	IF T_Data_ProcessImageLoadData.T_GeometryPara.arStartDiameter[6] <> T_Data_ProcessImageData.T_GeometryPara.arStartDiameter[6] THEN xProcessValueModified:=TRUE; RETURN; END_IF
	IF T_Data_ProcessImageLoadData.T_GeometryPara.arEndDiameter[6] <> T_Data_ProcessImageData.T_GeometryPara.arEndDiameter[6] THEN xProcessValueModified:=TRUE; RETURN; END_IF
	IF T_Data_ProcessImageLoadData.T_GeometryPara.arSectionLength[6] <> T_Data_ProcessImageData.T_GeometryPara.arSectionLength[6] THEN xProcessValueModified:=TRUE; RETURN; END_IF
	IF T_Data_ProcessImageLoadData.T_GeometryPara.arSectionPitch[6] <> T_Data_ProcessImageData.T_GeometryPara.arSectionPitch[6] THEN xProcessValueModified:=TRUE; RETURN; END_IF
	IF T_Data_ProcessImageLoadData.T_GeometryPara.axActiveSection[6] <> T_Data_ProcessImageData.T_GeometryPara.axActiveSection[6] THEN xProcessValueModified:=TRUE; RETURN; END_IF
(*09.12.2022: SOA *)
	IF T_Data_ProcessImageLoadData.T_PrismPara.rPrismaDistanceD1 <> T_Data_ProcessImageData.T_PrismPara.rPrismaDistanceD1 THEN xProcessValueModified:=TRUE; RETURN; END_IF
	IF T_Data_ProcessImageLoadData.T_PrismPara.rPrismaDistanceD2 <> T_Data_ProcessImageData.T_PrismPara.rPrismaDistanceD2 THEN xProcessValueModified:=TRUE; RETURN; END_IF
	IF T_Data_ProcessImageLoadData.T_PrismPara.rPrismaAngleA <> T_Data_ProcessImageData.T_PrismPara.rPrismaAngleA THEN xProcessValueModified:=TRUE; RETURN; END_IF
	IF T_Data_ProcessImageLoadData.T_PrismPara.bStateInputPrisma <> T_Data_ProcessImageData.T_PrismPara.bStateInputPrisma THEN xProcessValueModified:=TRUE; RETURN; END_IF
	IF T_Data_ProcessImageLoadData.T_PrismPara.rToolDiameterMin <> T_Data_ProcessImageData.T_PrismPara.rToolDiameterMin THEN xProcessValueModified:=TRUE; RETURN; END_IF
	IF T_Data_ProcessImageLoadData.T_PrismPara.rToolDiameterMax <> T_Data_ProcessImageData.T_PrismPara.rToolDiameterMax THEN xProcessValueModified:=TRUE; RETURN; END_IF
	IF T_Data_ProcessImageLoadData.T_PrismPara.rPrismaFactor <> T_Data_ProcessImageData.T_PrismPara.rPrismaFactor THEN xProcessValueModified:=TRUE; RETURN; END_IF

	IF T_Data_ProcessImageLoadData.T_ProcessPara.rOffsetBeforeToolDiaGrindFeedProcess <> T_Data_ProcessImageData.T_ProcessPara.rOffsetBeforeToolDiaGrindFeedProcess THEN xProcessValueModified:=TRUE; RETURN; END_IF
	IF T_Data_ProcessImageLoadData.T_ProcessPara.rSecurityPosGrindFeedProcess <> T_Data_ProcessImageData.T_ProcessPara.rSecurityPosGrindFeedProcess THEN xProcessValueModified:=TRUE; RETURN; END_IF
	IF T_Data_ProcessImageLoadData.T_ProcessPara.rSpeedBackwardGrindFeed <> T_Data_ProcessImageData.T_ProcessPara.rSpeedBackwardGrindFeed THEN xProcessValueModified:=TRUE; RETURN; END_IF
	IF T_Data_ProcessImageLoadData.T_ProcessPara.rSpeedForwardFastGrindFeed <> T_Data_ProcessImageData.T_ProcessPara.rSpeedForwardFastGrindFeed THEN xProcessValueModified:=TRUE; RETURN; END_IF
	IF T_Data_ProcessImageLoadData.T_ProcessPara.rSpeedForwardSlowGrindFeed <> T_Data_ProcessImageData.T_ProcessPara.rSpeedForwardSlowGrindFeed THEN xProcessValueModified:=TRUE; RETURN; END_IF
	IF xMicroRodActive THEN
		IF T_Data_ProcessImageLoadData.T_ProcessPara.rSpeedStartPosToolFeedProcess <> T_Data_ProcessImageData.T_ProcessPara.rSpeedStartPosToolFeedProcess THEN xProcessValueModified:=TRUE; RETURN; END_IF
		IF T_Data_ProcessImageLoadData.T_ProcessPara.rStartPosToolFeedAuto <> T_Data_ProcessImageData.T_ProcessPara.rStartPosToolFeedAuto THEN xProcessValueModified:=TRUE; RETURN; END_IF
	END_IF;
	IF T_Data_ProcessImageLoadData.T_ProcessPara.rToolDiameterProcess <> T_Data_ProcessImageData.T_ProcessPara.rToolDiameterProcess THEN xProcessValueModified:=TRUE; RETURN; END_IF
	IF T_Data_ProcessImageLoadData.T_ProcessPara.rToolTensionProcess <> T_Data_ProcessImageData.T_ProcessPara.rToolTensionProcess THEN xProcessValueModified:=TRUE; RETURN; END_IF

	IF T_Data_ProcessImageLoadData.T_AutoGeometryPara.iCycleGeometry <> T_Data_ProcessImageData.T_AutoGeometryPara.iCycleGeometry THEN xProcessValueModified:=TRUE; RETURN; END_IF
	IF xMicroRodActive THEN
		IF T_Data_ProcessImageLoadData.T_AutoGeometryPara.rPlungeCycleGrindFeedGeometry <> T_Data_ProcessImageData.T_AutoGeometryPara.rPlungeCycleGrindFeedGeometry THEN xProcessValueModified:=TRUE; RETURN; END_IF
	END_IF;
	IF T_Data_ProcessImageLoadData.T_AutoGeometryPara.rDisplaceLengthToolFeedGeometry <> T_Data_ProcessImageData.T_AutoGeometryPara.rDisplaceLengthToolFeedGeometry THEN xProcessValueModified:=TRUE; RETURN; END_IF
	IF T_Data_ProcessImageLoadData.T_AutoGeometryPara.rDisplaceSpeedGrindFeedGeometry <> T_Data_ProcessImageData.T_AutoGeometryPara.rDisplaceSpeedGrindFeedGeometry THEN xProcessValueModified:=TRUE; RETURN; END_IF
	IF T_Data_ProcessImageLoadData.T_AutoGeometryPara.rPlungeLengthToolFeedGeometry <> T_Data_ProcessImageData.T_AutoGeometryPara.rPlungeLengthToolFeedGeometry THEN xProcessValueModified:=TRUE; RETURN; END_IF
	IF T_Data_ProcessImageLoadData.T_AutoGeometryPara.rPlungeSpeedGrindFeedGeometry <> T_Data_ProcessImageData.T_AutoGeometryPara.rPlungeSpeedGrindFeedGeometry THEN xProcessValueModified:=TRUE; RETURN; END_IF
	IF T_Data_ProcessImageLoadData.T_AutoGeometryPara.rSpeedToolRotationGeometry <> T_Data_ProcessImageData.T_AutoGeometryPara.rSpeedToolRotationGeometry THEN xProcessValueModified:=TRUE; RETURN; END_IF
	IF T_Data_ProcessImageLoadData.T_AutoGeometryPara.xDisplaceActivationGeometry <> T_Data_ProcessImageData.T_AutoGeometryPara.xDisplaceActivationGeometry THEN xProcessValueModified:=TRUE; RETURN; END_IF
	IF T_Data_ProcessImageLoadData.T_AutoGeometryPara.xPlungeActivationGeometry <> T_Data_ProcessImageData.T_AutoGeometryPara.xPlungeActivationGeometry THEN xProcessValueModified:=TRUE; RETURN; END_IF

	IF T_Data_ProcessImageLoadData.T_AutoGroovePara.rDisplaceLengthToolFeedGroove <> T_Data_ProcessImageData.T_AutoGroovePara.rDisplaceLengthToolFeedGroove THEN xProcessValueModified:=TRUE; RETURN; END_IF
	IF T_Data_ProcessImageLoadData.T_AutoGroovePara.rDisplaceSpeedGrindFeedGroove <> T_Data_ProcessImageData.T_AutoGroovePara.rDisplaceSpeedGrindFeedGroove THEN xProcessValueModified:=TRUE; RETURN; END_IF
	IF T_Data_ProcessImageLoadData.T_AutoGroovePara.rPitchGroove <> T_Data_ProcessImageData.T_AutoGroovePara.rPitchGroove THEN xProcessValueModified:=TRUE; RETURN; END_IF
	IF T_Data_ProcessImageLoadData.T_AutoGroovePara.rPlungeLengthToolFeedGroove <> T_Data_ProcessImageData.T_AutoGroovePara.rPlungeLengthToolFeedGroove THEN xProcessValueModified:=TRUE; RETURN; END_IF
	IF T_Data_ProcessImageLoadData.T_AutoGroovePara.rPlungeSpeedGrindFeedGroove <> T_Data_ProcessImageData.T_AutoGroovePara.rPlungeSpeedGrindFeedGroove THEN xProcessValueModified:=TRUE; RETURN; END_IF
	IF T_Data_ProcessImageLoadData.T_AutoGroovePara.rSpeedToolRotationGroove <> T_Data_ProcessImageData.T_AutoGroovePara.rSpeedToolRotationGroove THEN xProcessValueModified:=TRUE; RETURN; END_IF
	IF T_Data_ProcessImageLoadData.T_AutoGroovePara.xDisplaceActivationGroove <> T_Data_ProcessImageData.T_AutoGroovePara.xDisplaceActivationGroove THEN xProcessValueModified:=TRUE; RETURN; END_IF
	IF T_Data_ProcessImageLoadData.T_AutoGroovePara.xPlungeActivationGroove <> T_Data_ProcessImageData.T_AutoGroovePara.xPlungeActivationGroove THEN xProcessValueModified:=TRUE; RETURN; END_IF
	IF T_Data_ProcessImageLoadData.T_AutoGroovePara.xBlockGrindFeeder <> T_Data_ProcessImageData.T_AutoGroovePara.xBlockGrindFeeder THEN xProcessValueModified:=TRUE; RETURN; END_IF
	IF T_Data_ProcessImageLoadData.T_AutoGroovePara.iNumberOfGrooves <> T_Data_ProcessImageData.T_AutoGroovePara.iNumberOfGrooves THEN xProcessValueModified:=TRUE; RETURN; END_IF
	IF T_Data_ProcessImageLoadData.T_AutoGroovePara.iSpeedGrindSpindle <> T_Data_ProcessImageData.T_AutoGroovePara.iSpeedGrindSpindle THEN xProcessValueModified:=TRUE; RETURN; END_IF

	IF T_Data_ProcessImageLoadData.T_CalibrationPara.rDisplaceLengthToolFeedCalib <> T_Data_ProcessImageData.T_CalibrationPara.rDisplaceLengthToolFeedCalib THEN xProcessValueModified:=TRUE; RETURN; END_IF
	IF T_Data_ProcessImageLoadData.T_CalibrationPara.rDisplaceSpeedGrindFeedCalib <> T_Data_ProcessImageData.T_CalibrationPara.rDisplaceSpeedGrindFeedCalib THEN xProcessValueModified:=TRUE; RETURN; END_IF
	IF NOT(xMicroRodActive) THEN
		IF T_Data_ProcessImageLoadData.T_CalibrationPara.rMeasureOffsetToolFeedCalib <> T_Data_ProcessImageData.T_CalibrationPara.rMeasureOffsetToolFeedCalib THEN xProcessValueModified:=TRUE; RETURN; END_IF
	END_IF;
	IF xMicroRodActive THEN
		IF T_Data_ProcessImageLoadData.T_CalibrationPara.rMeasurePosToolFeedCalib <> T_Data_ProcessImageData.T_CalibrationPara.rMeasurePosToolFeedCalib THEN xProcessValueModified:=TRUE; RETURN; END_IF
		IF T_Data_ProcessImageLoadData.T_CalibrationPara.rStartPosToolFeedCalib <> T_Data_ProcessImageData.T_CalibrationPara.rStartPosToolFeedCalib THEN xProcessValueModified:=TRUE; RETURN; END_IF
	END_IF;
	IF T_Data_ProcessImageLoadData.T_CalibrationPara.rPitchCalib <> T_Data_ProcessImageData.T_CalibrationPara.rPitchCalib THEN xProcessValueModified:=TRUE; RETURN; END_IF
	IF T_Data_ProcessImageLoadData.T_CalibrationPara.rPlungeLengthGrindFeedCalib <> T_Data_ProcessImageData.T_CalibrationPara.rPlungeLengthGrindFeedCalib THEN xProcessValueModified:=TRUE; RETURN; END_IF
	IF T_Data_ProcessImageLoadData.T_CalibrationPara.rPlungeLengthToolFeedCalib <> T_Data_ProcessImageData.T_CalibrationPara.rPlungeLengthToolFeedCalib THEN xProcessValueModified:=TRUE; RETURN; END_IF
	IF T_Data_ProcessImageLoadData.T_CalibrationPara.rPlungeSpeedGrindFeedCalib <> T_Data_ProcessImageData.T_CalibrationPara.rPlungeSpeedGrindFeedCalib THEN xProcessValueModified:=TRUE; RETURN; END_IF
	IF T_Data_ProcessImageLoadData.T_CalibrationPara.rSpeedToolRotationCalib <> T_Data_ProcessImageData.T_CalibrationPara.rSpeedToolRotationCalib THEN xProcessValueModified:=TRUE; RETURN; END_IF
	IF T_Data_ProcessImageLoadData.T_CalibrationPara.rToolLengthCylinderPartCalib <> T_Data_ProcessImageData.T_CalibrationPara.rToolLengthCylinderPartCalib THEN xProcessValueModified:=TRUE; RETURN; END_IF
	IF T_Data_ProcessImageLoadData.T_CalibrationPara.xDisplaceActivationCalib <> T_Data_ProcessImageData.T_CalibrationPara.xDisplaceActivationCalib THEN xProcessValueModified:=TRUE; RETURN; END_IF
	IF T_Data_ProcessImageLoadData.T_CalibrationPara.xPlungeActivationCalib <> T_Data_ProcessImageData.T_CalibrationPara.xPlungeActivationCalib THEN xProcessValueModified:=TRUE; RETURN; END_IF
END_FUNCTION_BLOCK

(* POU PRG_VISU_LAYER5/FB_VISU/FB_CALC_TORQUE, ST *)
FUNCTION_BLOCK FB_CALC_TORQUE
VAR_INPUT
	xStart:BOOL;				(* start the calculation of the mean value of the torque *)
	uiActualTorque:UINT;		(* actual current value *)
	uiZeroTorque:UINT;		(* set value of the current value for scale the range *)
	iStepCalc:INT;			(* number of mean value *)
END_VAR
VAR_OUTPUT
	uiCalcTorque:UINT;		(* calculated torque value in % of the maximal torque of the motor *)
END_VAR
VAR
	auiSaveTorque: ARRAY [1..200] OF UINT;
	auiTmpSaveTorque: ARRAY [1..200] OF UINT;
	auiDeleteTorque: ARRAY [1..200] OF UINT;
	uiSumTorque: UINT;
	ii: INT;
	xInit: BOOL;
	uiTmpZeroTorque:UINT;
	rMaxMotorCurrent: REAL;
	rMaxMotorTorque: REAL;
END_VAR
(****************************************************************************************************************************************************)
(***********             This Functionblock calc the torque of the ToolRotation with set and reset torque function                         ************)
(****************************************************************************************************************************************************)
uiCalcTorque:=0;
IF NOT(xStart) AND xInit THEN
	xInit:=FALSE;
	auiSaveTorque:=auiDeleteTorque;
	auiTmpSaveTorque:=auiDeleteTorque;
	uiTmpZeroTorque:=uiZeroTorque;
END_IF;
IF xStart THEN
	xInit:=TRUE;
	uiSumTorque:=0;
	IF (uiZeroTorque <> uiTmpZeroTorque) THEN
		auiSaveTorque:=auiDeleteTorque;
		auiTmpSaveTorque:=auiDeleteTorque;
		uiTmpZeroTorque:=uiZeroTorque;
	END_IF;
	IF (iStepCalc > 0) AND (iStepCalc <= 200) THEN
		FOR ii:=1 TO (iStepCalc - 1)  DO
			auiTmpSaveTorque[ii+1]:=auiSaveTorque[ii];
			uiSumTorque:=uiSumTorque + auiSaveTorque[ii];
		END_FOR;
		auiSaveTorque:=auiTmpSaveTorque;
		IF (uiTmpZeroTorque <= uiActualTorque) THEN
			auiSaveTorque[1]:=uiActualTorque - uiTmpZeroTorque;
		ELSE
			auiSaveTorque[1]:=0;
		END_IF;
		uiSumTorque:=uiSumTorque + auiSaveTorque[1];
		uiSumTorque:=uiSumTorque/iStepCalc;
		rMaxMotorCurrent:=6.0;	(* EcoStep Motor 23S21  *)
		rMaxMotorTorque:=(rMaxMotorCurrent * 0.16) * 1000.0;	(* 0.16 = 0.16Nm/A -->1000.0= Umwandlung in mNm *)
		uiCalcTorque:=REAL_TO_UINT((UINT_TO_REAL(uiSumTorque) / (REAL_TO_UINT(rMaxMotorTorque) - uiTmpZeroTorque)) * 100.0);	(* Ausgabe in % des Max Stromes *)
		IF (uiCalcTorque >= 100) THEN
			uiCalcTorque:=100;
		END_IF;
	END_IF;
END_IF;
END_FUNCTION_BLOCK

(* POU PRG_VISU_LAYER5/FB_VISU/FBQVIS_ERROR_LIST, ST *)
FUNCTION_BLOCK FBQVIS_ERROR_LIST
VAR_INPUT
	T_ErrorList:ST_ERROR_LIST;					(* Static define Error List *)
	T_ErrorNrList:ST_RETAIN_ERROR_DATA;		(* Daten welche im NOVram abgelegt sind *)
END_VAR
VAR_IN_OUT
	T_MsgErrorEnglish:ST_EXCHG_MESSAGE_ERROR;	(* Daten die auf der Visu in der Errorliste visualisiert werden *)
	T_MsgErrorDeutsch:ST_EXCHG_MESSAGE_ERROR;	(* Daten die auf der Visu in der Errorliste visualisiert werden *)
	T_MsgErrorFrancais:ST_EXCHG_MESSAGE_ERROR;	(* Daten die auf der Visu in der Errorliste visualisiert werden *)
END_VAR
VAR_OUTPUT
END_VAR
VAR
	FBErrorMessage:FB_ErrorMessage;
	ii:INT;
	diErrorNr: DINT;
	sErrorTimeStamp: STRING(12);
END_VAR
(****************************************************************************************************************************************************)
(***********                              This Functionblock fills the errorlist with the errormesse and the timestamp                                  ************)
(****************************************************************************************************************************************************)
	FOR ii:=1 TO 20 DO
		diErrorNr:=T_ErrorNrList.adiErrorListMachine[ii];
		sErrorTimeStamp:=T_ErrorNrList.asErrorTimeStampMachine[ii];
		sErrorTimeStamp:=CONCAT(sErrorTimeStamp,'--');
		IF (diErrorNr <> 0) THEN
			FBErrorMessage(	diErrorNr:=diErrorNr ,
							T_ErrorList:=T_ErrorList);
			T_MsgErrorEnglish.asMsgErrorList[ii]:=CONCAT(sErrorTimeStamp,FBErrorMessage.sErrorTextEnglish);
			T_MsgErrorDeutsch.asMsgErrorList[ii]:=CONCAT(sErrorTimeStamp,FBErrorMessage.sErrorTextDeutsch);
			T_MsgErrorFrancais.asMsgErrorList[ii]:=CONCAT(sErrorTimeStamp,FBErrorMessage.sErrorTextFrancais);
		ELSE
			T_MsgErrorEnglish.asMsgErrorList[ii]:='                                                                    ';
			T_MsgErrorDeutsch.asMsgErrorList[ii]:='                                                                    ';
			T_MsgErrorFrancais.asMsgErrorList[ii]:='                                                                    ';
		END_IF;
	END_FOR;
END_FUNCTION_BLOCK

(* POU PRG_VISU_LAYER5/FB_VISU/FB_SETERRORLIST, ST *)
FUNCTION_BLOCK FB_SETERRORLIST
VAR_INPUT
	TControlStation : ST_CONTROL;					(* Control structur of the data station structure *)
	TProcess : ST_PROCESS;						(* data structure of the processlevel *)
END_VAR
VAR_IN_OUT
	xParameterSaved:BOOL;						(* state, if the changed errorlist was saved *)
	T_ErrorNrList:ST_RETAIN_ERROR_DATA;		(* Daten welche im NOVram abgelegt sind *)
	xSetForceError:BOOL;							(* manual input of an error into the error list *)
	diSetForceErrorNr:DINT;						(* manual input of an error number into the error list *)
END_VAR
VAR_OUTPUT
	xSaveParameter:BOOL;						(* save the maked or updated error list into the Novram *)
END_VAR
VAR
	xTmpStation: BOOL;
	xTmpProcess: BOOL;
	iTmpStationNr:INT;
	xBlockProcessProc: BOOL;
	xBlockStationProc: BOOL;
	adiTmpErrorList: ARRAY [1..20] OF DINT;
	asTmpErrorList: ARRAY [1..20] OF STRING(12);
	ii:INT;
	xDataChanged: BOOL;
	xQuitError: BOOL;
	TimerCheckQuitError:TON;
	FBNT_GetTime:NT_GetTime;
	xUpdateProcTimeStamp:BOOL;
	xInitGetTime: BOOL;
END_VAR
(****************************************************************************************************************************************************)
(***********                       This Functionblock manage the machine error, for make and update the errorlist                             ************)
(****************************************************************************************************************************************************)
xTmpStation:=TControlStation.xError AND TControlStation.xActiveStation;
xTmpProcess:=TProcess.xError AND TProcess.xRdy;

IF NOT(xDataChanged) THEN
	IF NOT(TProcess.xEnd) AND TProcess.xError AND NOT(xBlockProcessProc) AND NOT(xBlockStationProc) AND NOT(xSetForceError) THEN
		xBlockProcessProc:=TRUE;
		iTmpStationNr:=0;
	END_IF;
	IF TProcess.xEnd AND xTmpStation AND NOT(xBlockStationProc) AND NOT(xBlockProcessProc) AND NOT(xSetForceError) THEN
		xBlockStationProc:=TRUE;
		iTmpStationNr:=1;
	END_IF;
	IF xBlockProcessProc AND NOT(xQuitError) THEN
		adiTmpErrorList:=T_ErrorNrList.adiErrorListMachine;
		T_ErrorNrList.adiErrorListMachine[1]:=TProcess.diErrorNr;
		FOR ii:=2 TO 20 DO
			T_ErrorNrList.adiErrorListMachine[ii]:=adiTmpErrorList[ii-1];
		END_FOR;
		xUpdateProcTimeStamp:=TRUE;
	END_IF;
	
	IF xBlockStationProc AND NOT(xQuitError) THEN
		adiTmpErrorList:=T_ErrorNrList.adiErrorListMachine;
		T_ErrorNrList.adiErrorListMachine[1]:=TControlStation.diErrorNr;
		FOR ii:=2 TO 20 DO
			T_ErrorNrList.adiErrorListMachine[ii]:=adiTmpErrorList[ii-1];
		END_FOR;
		xUpdateProcTimeStamp:=TRUE;
	END_IF;
	
	IF xSetForceError AND NOT(xQuitError) AND NOT(xBlockStationProc) AND NOT(xBlockProcessProc) THEN
		adiTmpErrorList:=T_ErrorNrList.adiErrorListMachine;
		T_ErrorNrList.adiErrorListMachine[1]:=diSetForceErrorNr;
		FOR ii:=2 TO 20 DO
			T_ErrorNrList.adiErrorListMachine[ii]:=adiTmpErrorList[ii-1];
		END_FOR;
		xUpdateProcTimeStamp:=TRUE;
		xSetForceError:=FALSE;
	ELSE
		xSetForceError:=FALSE;
	END_IF;

	IF xUpdateProcTimeStamp THEN
		IF NOT(xInitGetTime) THEN
			xInitGetTime:=TRUE;
			FBNT_GetTime(	NETID:= '',
							START:=FALSE );
		END_IF;
		FBNT_GetTime(	NETID:= '',
						START:= TRUE,
						TMOUT:= T#2s);
		IF NOT(FBNT_GetTime.BUSY) OR FBNT_GetTime.ERR THEN
			IF xUpdateProcTimeStamp THEN
				asTmpErrorList:=T_ErrorNrList.asErrorTimeStampMachine;
				IF NOT(FBNT_GetTime.ERR) THEN
					T_ErrorNrList.asErrorTimeStampMachine[1]:=Fct_ConvertDateToString(2,FBNT_GetTime.TIMESTR);
				ELSE
					T_ErrorNrList.asErrorTimeStampMachine[1]:='00.00 00:00';	(* Fehler beim lesen der Systemzeit, daher wird ein default-Wert gesetzt *)
				END_IF;
				FOR ii:=2 TO 20 DO
					T_ErrorNrList.asErrorTimeStampMachine[ii]:=asTmpErrorList[ii-1];
				END_FOR;
			END_IF;
			xInitGetTime:=FALSE;
			xUpdateProcTimeStamp:=FALSE;
			xDataChanged:=TRUE;
		END_IF;
	END_IF;
END_IF;

IF xBlockProcessProc OR xBlockStationProc THEN
	xQuitError:=TRUE;
	IF TControlStation.xQuitError OR TProcess.xQuitError THEN
		xBlockProcessProc:=xBlockStationProc:=xSetForceError:=xQuitError:=FALSE;
	END_IF;
	IF NOT(xTmpStation) AND NOT(xTmpProcess) THEN
		TimerCheckQuitError(IN:=TRUE,PT:=T#1s);
		IF TimerCheckQuitError.Q THEN
			TimerCheckQuitError(IN:=FALSE);
			xBlockProcessProc:=xBlockStationProc:=xSetForceError:=xQuitError:=FALSE;
		END_IF;
	ELSE
		TimerCheckQuitError(IN:=FALSE);
	END_IF;
ELSE
	xQuitError:=FALSE;
END_IF;

IF xDataChanged THEN
	xSaveParameter:=TRUE;
	IF xParameterSaved THEN
		xParameterSaved:=xDataChanged:=xSaveParameter:=FALSE;
	END_IF;
END_IF;
END_FUNCTION_BLOCK

(* POU PRG_PROCESS_LAYER4/FB_PROCESS/Fct_ConvertDateToString, ST *)
FUNCTION Fct_ConvertDateToString : STRING
VAR_INPUT
		iFormat:INT;	(* 0=Langes Date-Time Format; 1=Kurzes Date-Time Format; 2=Sehr Kurzes Date-Time Format *)
					(* 0='28.March 2007  08:47:01' *)
					(* 1='28.03.07 08:47' *)
					(* 2='28.03 08:47' *)
		TProcTimeStart:TIMESTRUCT;
END_VAR
VAR
	sTmpData:STRING(255);
	sTmpData1:STRING(255);
	wYear: WORD;
END_VAR
(****************************************************************************************************************************************************)
(***********                                This Functionblock formate a Date and Time String DD:MM HH:MM:SS                                     ************)
(****************************************************************************************************************************************************)
sTmpData:=sTmpData1:='';
IF (iFormat < 0) OR (iFormat > 2) THEN
	sTmpData1:='Wrong Date';
	Fct_ConvertDateToString:=sTmpData1;
	RETURN;
END_IF;
IF (TProcTimeStart.wDay <> 0) THEN
	IF (TProcTimeStart.wDay >= 0) AND (TProcTimeStart.wDay <= 9) THEN
		sTmpData1:=MUX(TProcTimeStart.wDay,'00','01','02','03','04','05','06','07','08','09');
		sTmpData:=CONCAT(sTmpData,sTmpData1);
	ELSE
		sTmpData:=CONCAT(sTmpData,WORD_TO_STRING(TProcTimeStart.wDay));
	END_IF;
	sTmpData:=CONCAT(sTmpData,'.');
ELSE
	sTmpData1:='Wrong Date';
	Fct_ConvertDateToString:=sTmpData1;
	RETURN;
END_IF;
IF (TProcTimeStart.wMonth <> 0) THEN
	IF (iFormat = 0) THEN
		sTmpData1:=MUX(TProcTimeStart.wMonth-1,'January','February','March','April','May','June','July','August','September','October','November','December');
	END_IF;
	IF (iFormat = 1) OR (iFormat = 2) THEN
		sTmpData1:=MUX(TProcTimeStart.wMonth-1,'01','02','03','04','05','06','07','08','09','10','11','12');
	END_IF;
ELSE
	sTmpData1:='Wrong Date';
	Fct_ConvertDateToString:=sTmpData1;
	RETURN;
END_IF;
sTmpData:=CONCAT(sTmpData,sTmpData1);
IF (iFormat = 0) THEN
	sTmpData:=CONCAT(sTmpData,' ');
END_IF;
IF (iFormat = 1) THEN
	sTmpData:=CONCAT(sTmpData,'.');
END_IF;
IF (iFormat = 2) THEN
	sTmpData:=CONCAT(sTmpData,' ');
END_IF;
IF (iFormat = 0) OR (iFormat = 1) THEN
	IF (TProcTimeStart.wYear <> 0) THEN
		IF (iFormat = 0) THEN
			sTmpData:=CONCAT(sTmpData,WORD_TO_STRING(TProcTimeStart.wYear));
			sTmpData:=CONCAT(sTmpData,'  ');
		END_IF;
		IF (iFormat = 1) THEN
			IF (TProcTimeStart.wYear >= 1000) AND (TProcTimeStart.wYear < 2000) THEN
				wYear:=TProcTimeStart.wYear - 1000;
			END_IF;
			IF (TProcTimeStart.wYear >= 2000) AND (TProcTimeStart.wYear < 3000) THEN
				wYear:=TProcTimeStart.wYear - 2000;
			END_IF;
			IF (wYear >= 0) AND (wYear < 10) THEN
				sTmpData1:=MUX(wYear,'00','01','02','03','04','05','06','07','08','09');
				sTmpData:=CONCAT(sTmpData,sTmpData1);
			ELSE
				sTmpData:=CONCAT(sTmpData,WORD_TO_STRING(wYear));
			END_IF;
			sTmpData:=CONCAT(sTmpData,' ');
		END_IF;
	ELSE
		sTmpData1:='Wrong Date';
		Fct_ConvertDateToString:=sTmpData1;
		RETURN;
	END_IF;
END_IF;
IF (TProcTimeStart.wHour >= 0) AND (TProcTimeStart.wHour <= 9) THEN
	sTmpData1:=MUX(TProcTimeStart.wHour,'00','01','02','03','04','05','06','07','08','09');
	sTmpData:=CONCAT(sTmpData,sTmpData1);
ELSE
	sTmpData:=CONCAT(sTmpData,WORD_TO_STRING(TProcTimeStart.wHour));
END_IF;
sTmpData:=CONCAT(sTmpData,':');
IF (TProcTimeStart.wMinute >= 0) AND (TProcTimeStart.wMinute <= 9) THEN
	sTmpData1:=MUX(TProcTimeStart.wMinute,'00','01','02','03','04','05','06','07','08','09');
	sTmpData:=CONCAT(sTmpData,sTmpData1);
ELSE
	sTmpData:=CONCAT(sTmpData,WORD_TO_STRING(TProcTimeStart.wMinute));
END_IF;
IF (iFormat = 0) THEN
	sTmpData:=CONCAT(sTmpData,':');
	IF (TProcTimeStart.wSecond >= 0) AND (TProcTimeStart.wSecond <= 9) THEN
		sTmpData1:=MUX(TProcTimeStart.wSecond,'00','01','02','03','04','05','06','07','08','09');
		sTmpData:=CONCAT(sTmpData,sTmpData1);
	ELSE
		sTmpData:=CONCAT(sTmpData,WORD_TO_STRING(TProcTimeStart.wSecond));
	END_IF;
END_IF;
Fct_ConvertDateToString:=sTmpData;
END_FUNCTION

(* POU PRG_VISU_LAYER5/FB_VISU/FBQVIS_CLEARERROR, ST *)
FUNCTION_BLOCK FBQVIS_CLEARERROR
VAR_INPUT
	xExecute:BOOL;				(* quit the error *)
	iError:INT;					(* occured error number *)
END_VAR
VAR_IN_OUT
	T_Message:ST_EXCHG_MESSAGE;		(* data structure for the message handling *)
	T_Station:ST_STATION;				(* data structure for the stationlevel *)
	T_Process : ST_PROCESS;			(* data structure for the processlevel *)
	T_NovRAM:ST_NOVRAM;				(* data structure for the Novram *)
	T_Profile:ST_PROFILE;				(* data structure for the profile management *)
	T_HDD:ST_HDD;						(* data structure for the file management *)
END_VAR
VAR_OUTPUT
	xDone:BOOL;
	xNotReady:BOOL;
	xErr:BOOL;
	udiErrorID:UDINT;
END_VAR
VAR
(* Trigger *)
	RisingEdgeExecute:R_TRIG;
(* Pointer *)
	ptrActivStation:POINTER TO ST_STATION;
(* Variable *)
	xClearError_Done:BOOL;
	xClearError_Err:BOOL;
	xClearError_NotReady:BOOL;
	xStepClearDone:BOOL;
	udiClearError_ErrorID:UDINT;
	iStepClearErrorStation:INT;
	iStepClearErrorMachine:INT;
	iStepClearStandardError: INT;
	xClearProcess:BOOL;
	xClearStation:BOOL;
	xClearStandardError:BOOL;
	xClearConifgErrStation: BOOL;
	xTmp: BOOL;
	xClearAxis: BOOL;
	iStepClearErrorAxis: INT;
	xTmp1: BOOL;
	xActiveMicroRod: BOOL;
	iTryAgain: INT;
END_VAR
(****************************************************************************************************************************************************)
(***********              This Functionblock manage an occured machine error so that the right component are quittet              ************)
(****************************************************************************************************************************************************)
	IF (T_NovRAM.T_Data.T_Standard.T_MachineConfig.iConfigMachineType = 2) THEN
		xActiveMicroRod:=TRUE;
	ELSE
		xActiveMicroRod:=FALSE;
	END_IF;

	RisingEdgeExecute(CLK:=xExecute);
	IF RisingEdgeExecute.Q THEN
	(* Init. variable by start clear error *)
		(* ...output *)
		xDone:=FALSE;
		xNotReady:=FALSE;
		xErr:=FALSE;
		udiErrorID:=16#0;
		(* ...variable *)
		xClearError_Done:=FALSE;
		xClearError_Err:=FALSE;
		xClearError_NotReady:=FALSE;
		xStepClearDone:=FALSE;
		iStepClearErrorStation:=1;
		iStepClearErrorMachine:=1;
		iStepClearStandardError:=1;
		iStepClearErrorAxis:=1;
		(* determin clear action *)
		xClearProcess:=xClearStation:=xClearAxis:=xClearStandardError:=FALSE;
		xClearConifgErrStation:=FALSE;
		IF T_Process.xError THEN
			xClearProcess:=TRUE;
		ELSE
			IF T_Station.TControl.xError AND NOT(T_Station.TControl.xEnd) THEN ptrActivStation:=ADR(T_Station); xClearStation:=TRUE; END_IF
			xTmp:=	(T_Station.THardware.TAxisToolLeft.T_CtrleSingle.xErr OR
					(T_Station.THardware.TAxisToolCenter.T_CtrleSingle.xErr AND xActiveMicroRod) OR
					T_Station.THardware.TAxisToolRight.T_CtrleSingle.xErr OR
					T_Station.THardware.TAxisToolFeeder.T_CtrleSingle.xErr OR
					T_Station.THardware.TAxisGrindFeeder.T_CtrleSingle.xErr) AND
					NOT(xClearStation);
			IF xTmp THEN
				xClearAxis:=TRUE;
			END_IF;
			IF T_Station.TControl.xError AND T_Station.TControl.xEnd AND NOT(xClearAxis) THEN
				xClearConifgErrStation:=TRUE;
			END_IF
		END_IF
		IF NOT xClearProcess AND NOT xClearStation AND NOT xClearConifgErrStation AND NOT xClearAxis THEN xClearStandardError:=TRUE; END_IF
		(* Exit FB *)
		RETURN;
	END_IF

	IF xClearProcess THEN
	(* Reset Error machine *)
		CASE iStepClearErrorMachine OF
		(* check station *)
		1:	IF T_Process.xError THEN iStepClearErrorMachine:=10; ELSE iStepClearErrorMachine:=90; END_IF
		(* activ clear error *)
		10:	T_Process.xQuitError:=TRUE;
			(* next step *)
			iStepClearErrorMachine:=20;
			xStepClearDone:=FALSE;
		(* waiting end clearing error *)
		20:	IF NOT T_Process.xQuitError THEN
				iStepClearErrorMachine:=90;
				xStepClearDone:=FALSE;
			END_IF
			IF T_Process.xError THEN iStepClearErrorMachine:=90; END_IF
		(* Clear error station done *)
		90:	xClearError_Done:=TRUE;
		(* Error *)
		99:	xClearError_Err:=TRUE;
		END_CASE
	END_IF

	IF xClearStation THEN
	(* Reset Error station *)
		CASE iStepClearErrorStation OF
		(* check station *)
		1:	IF ptrActivStation^.TControl.xError THEN iStepClearErrorStation:=10;
			ELSE IStepClearErrorStation:=90; END_IF
		(* activ clear error *)
		10:	ptrActivStation^.TControl.xQuitError:=TRUE;
			(* next step *)
			iStepClearErrorStation:=20;
			xStepClearDone:=FALSE;
		(* waiting end clearing error *)
		20:	IF NOT(xStepClearDone) THEN
			(* release action *)
				ptrActivStation^.TControl.xQuitError:=FALSE;
				xStepClearDone:=TRUE;
			ELSE
				IF ptrActivStation^.TControl.xEnd THEN
				(* confirm clear error, next step *)
					iStepClearErrorStation:=90;
					xStepClearDone:=FALSE;
				END_IF
				IF ptrActivStation^.TControl.xError THEN iStepClearErrorStation:=99; END_IF
			END_IF
		(* Clear error station done *)
		90:	xClearError_Done:=TRUE;
		(* Error *)
		99:	xClearError_Done:=TRUE;
		END_CASE
	END_IF

	IF xClearConifgErrStation THEN
		T_Station.TControl.xError:=FALSE;
		xClearConifgErrStation:=FALSE;
		(* Clear error station done *)
		xClearError_Done:=TRUE;
	END_IF;

	IF xClearAxis THEN
	(* Reset Error axis *)
		CASE iStepClearErrorAxis OF
		(* check station *)
		1:	xTmp:=	T_Station.THardware.TAxisToolLeft.T_CtrleSingle.xErr OR
					(T_Station.THardware.TAxisToolCenter.T_CtrleSingle.xErr AND xActiveMicroRod) OR
					T_Station.THardware.TAxisToolRight.T_CtrleSingle.xErr OR
					T_Station.THardware.TAxisToolFeeder.T_CtrleSingle.xErr OR
					T_Station.THardware.TAxisGrindFeeder.T_CtrleSingle.xErr;
			IF xTmp THEN iStepClearErrorAxis:=10;
			ELSE iStepClearErrorAxis:=90; END_IF
			iTryAgain:=0;
		(* activ clear error *)
		10:	T_Station.THardware.TAxisToolLeft.T_CtrleSingle.iFunction:=1;
			T_Station.THardware.TAxisToolLeft.T_CtrleSingle.xExecute:=T_Station.THardware.TAxisToolLeft.T_CtrleSingle.xErr;
			IF xActiveMicroRod THEN
				T_Station.THardware.TAxisToolCenter.T_CtrleSingle.iFunction:=1;
				T_Station.THardware.TAxisToolCenter.T_CtrleSingle.xExecute:=T_Station.THardware.TAxisToolCenter.T_CtrleSingle.xErr;
			END_IF;
			T_Station.THardware.TAxisToolRight.T_CtrleSingle.iFunction:=1;
			T_Station.THardware.TAxisToolRight.T_CtrleSingle.xExecute:=T_Station.THardware.TAxisToolRight.T_CtrleSingle.xErr;
			T_Station.THardware.TAxisToolFeeder.T_CtrleSingle.iFunction:=1;
			T_Station.THardware.TAxisToolFeeder.T_CtrleSingle.xExecute:=T_Station.THardware.TAxisToolFeeder.T_CtrleSingle.xErr;
			T_Station.THardware.TAxisGrindFeeder.T_CtrleSingle.iFunction:=1;
			T_Station.THardware.TAxisGrindFeeder.T_CtrleSingle.xExecute:=T_Station.THardware.TAxisGrindFeeder.T_CtrleSingle.xErr;
			(* next step *)
			iStepClearErrorAxis:=20;
			xStepClearDone:=FALSE;
		(* waiting end clearing error *)
		20:	IF NOT(xStepClearDone) THEN
			(* release action *)
				xStepClearDone:=TRUE;
			ELSE
				xTmp:=	T_Station.THardware.TAxisToolLeft.T_CtrleSingle.xDone AND
						((T_Station.THardware.TAxisToolCenter.T_CtrleSingle.xDone AND xActiveMicroRod) OR NOT(xActiveMicroRod)) AND
						T_Station.THardware.TAxisToolRight.T_CtrleSingle.xDone AND
						T_Station.THardware.TAxisToolFeeder.T_CtrleSingle.xDone AND
						T_Station.THardware.TAxisGrindFeeder.T_CtrleSingle.xDone;
				xTmp1:=	T_Station.THardware.TAxisToolLeft.T_CtrleSingle.xErr OR
						(T_Station.THardware.TAxisToolCenter.T_CtrleSingle.xErr AND xActiveMicroRod) OR
						T_Station.THardware.TAxisToolRight.T_CtrleSingle.xErr OR
						T_Station.THardware.TAxisToolFeeder.T_CtrleSingle.xErr OR
						T_Station.THardware.TAxisGrindFeeder.T_CtrleSingle.xErr;
				IF xTmp THEN
				(* confirm clear error, next step *)
					iStepClearErrorAxis:=90;
					xStepClearDone:=FALSE;
				END_IF
				IF xTmp1 THEN
					iTryAgain:=iTryAgain + 1;
					IF (iTryAgain <= 3) THEN
						(* Reset maximal three times *)
						iStepClearErrorAxis:=10;
					ELSE
						iStepClearErrorAxis:=99;
					END_IF;
				END_IF

			END_IF
		(* Clear error station done *)
		90:	xClearError_Done:=TRUE;
		(* Error *)
		99:	xClearError_Done:=TRUE;
		END_CASE;
	END_IF;

	IF xClearStandardError THEN
	(* Reset Error standard *)
		CASE iStepClearStandardError OF
		(* check NovRAM state *)
		1:	iStepClearStandardError:=10;
			IF T_NovRAM.T_Ctrle.xErr THEN T_NovRAM.T_Ctrle.xReset:=TRUE; END_IF
		(* check Profile State *)
		10:	iStepClearStandardError:=20;
			IF T_Profile.T_Ctrle.xErr THEN T_Profile.T_Ctrle.xReset:=TRUE; END_IF
		(* check HDD state *)
		20:	iStepClearStandardError:=90;
			IF T_HDD.T_Ctrle.xErr THEN T_HDD.T_Ctrle.xReset:=TRUE; END_IF
		(* Clear error station done *)
		90:	xClearError_Done:=TRUE;
		END_CASE
	END_IF

(* FB Done/Err/NotReady *)
	IF xClearError_Done OR xClearError_Err OR xClearError_NotReady THEN
	(* copy value *)
		T_Message.iState:=0;
		T_Message.sDynamicTextEnglish:='';
		T_Message.sDynamicTextDeutsch:='';
		T_Message.sDynamicTextFrancais:='';
		xDone:=xClearError_Done;
		xNotReady:=xClearError_NotReady;
		xErr:=FALSE;
		udiErrorID:=udiClearError_ErrorID;
		(* Init. function state *)
		xClearProcess:=FALSE;
		xClearStation:=FALSE;
		xClearAxis:=FALSE;
		xClearStandardError:=FALSE;
		xClearConifgErrStation:=FALSE;
	END_IF
END_FUNCTION_BLOCK

(* POU GENERAL/FB_CALCPROCESSTIME, ST *)
FUNCTION_BLOCK FB_CALCPROCESSTIME
VAR_INPUT
	T_Geometry:ST_GEOMETRY;									(* Structure of the NovRAM parameter *)
	T_AutoGeometryPara:ST_EXCHG_PARAM_AUTOGEOMETRY;		(* Structure of the NovRAM parameter *)
	T_CalibrationPara:ST_EXCHG_PARAM_CALIBRATION;			(* Structure of the NovRAM parameter *)
	T_AutoGroovePara:ST_EXCHG_PARAM_AUTOGROOVE;			(* Structure of the NovRAM parameter *)
	T_ProcessPara:ST_EXCHG_PARAM_PROCESS;					(* Structure of the NovRAM parameter *)
	rToolRotationSpeed:REAL;										(* Speed of the ToolRotation in U/Min *)
	rToolDiameter:REAL;											(* Diameter of the Tool in um *)
	rToolDiameterWithOffset:REAL;			(* diameter of the unworked Tool plus the offset for plunge and displace procedure *)
	iAutoProcess:INT;												(* 0=Calibration, 1=AutoGeometry process, 2=AutoGroove process *)
	xMicroRodActive:BOOL;										(* choice of the machine MicroWire or MicroRod *)
END_VAR
VAR_IN_OUT
	T_WorkTool:ST_WORKTOOL;									(* Tool parameter *)
END_VAR
VAR_OUTPUT
	rProcessTime: REAL;											(* calculated process time *)
END_VAR
VAR
	FBToolCalcul:FB_TOOL_CALCUL;
	ii: INT;
	rTimeLeftWork: REAL;
	iStartSection: INT;
	iEndSection: INT;
	rPlungeGrind: REAL;
	rDisplaceGrind: REAL;
	rGrindFeederPlunge: REAL;
	xResetFB: BOOL;
	xInitFB:BOOL;
(*11.10.2010 KFS {	*)
	FBCalcPlungeGrinding: FB_CALC_PLUNGE_GRINDING;
	FBCalcPlungeGrindingMultiCycle: FB_CALC_PLUNGE_GRINDING_MultiCycle;
(*11.10.2010 KFS }	*)
	rPlungeCycleGrindFeedGeometry: REAL;
	iTmpStartSection: INT;
	xCalculation: BOOL;
	rToolFeedLength: REAL;
	rSpeedToolFeed: REAL;
	rTimeAddLeftWork:REAL;
	rToolLength:REAL;
	rPlungeGrind2: REAL;
	rTimeAddLeftWorkPlungeGrind: REAL;
	rTimeAddLeftWorkPlungeGrind2: REAL;
	rTimeAddLeftWorkToolFeed: REAL;
END_VAR
(****************************************************************************************************************************************************)
(***********        This Functionblock calculates the time,  needed to work a geometry, groove or  calibration      		    ************)
(****************************************************************************************************************************************************)
	rProcessTime:=0.0;
	rTimeLeftWork:=0;
	iStartSection:=0;
	iEndSection:=0;
	xInitFB:=FALSE;
	IF (iAutoProcess = 1) THEN
	(* calculate the time for the process AutoGeometry or AutoGroove *)
		T_WorkTool.iTotalCountDownPlungeCycle:=0;
		(* Check Start and End Section of the ToolGeometry *)
		FOR ii:=1 TO 6 DO
			IF T_Geometry.axActiveSection[ii] THEN
				IF (iStartSection = 0) THEN
					iStartSection:=ii;
				END_IF;
				iEndSection:=ii;
			END_IF;
		END_FOR;
		xResetFB:=TRUE;
		(* reset first the FB for calculate the grinding plunge for each sections *)
		FBCalcPlungeGrindingMultiCycle(	rToolDiameter:= rToolDiameter,
										rToolDiameterWithOffset:=rToolDiameterWithOffset,
										xReset:= xResetFB,
										xInit:=xInitFB);
		xInitFB:=TRUE;
		FBCalcPlungeGrindingMultiCycle(	T_Geometry:= T_Geometry,
										T_AutoGeometryPara:= T_AutoGeometryPara,
										rToolDiameter:= rToolDiameter,
										rToolDiameterWithOffset:=rToolDiameterWithOffset,
										rPlungeCycleGrindFeedGeometry:=rPlungeCycleGrindFeedGeometry,
										iStartSection:= iStartSection,
										iEndSection:= iEndSection,
										xReset:= xResetFB,
										xInit:=xInitFB);

		rPlungeCycleGrindFeedGeometry:=1.0;
		IF (iAutoProcess = 1) AND xMicroRodActive THEN
			rPlungeCycleGrindFeedGeometry:=T_AutoGeometryPara.rPlungeCycleGrindFeedGeometry;
		END_IF;
		T_WorkTool.rToolRotationSpeed:=rToolRotationSpeed;
		xCalculation:=TRUE;
		WHILE(xCalculation) DO
			(* calculate the grinding way of each section *)
			FBCalcPlungeGrindingMultiCycle(	T_Geometry:= T_Geometry,
											T_AutoGeometryPara:= T_AutoGeometryPara,
											rToolDiameter:= rToolDiameter,
											rToolDiameterWithOffset:=rToolDiameterWithOffset,
											rPlungeCycleGrindFeedGeometry:=rPlungeCycleGrindFeedGeometry,
											iStartSection:= iStartSection,
											iEndSection:= iEndSection,
											xReset:= xResetFB,
											xInit:=xInitFB);
			IF FBCalcPlungeGrindingMultiCycle.xEndWorking THEN		(* check if the end of the to work Tool is reached *)
				xCalculation:=FALSE;
				EXIT;
			END_IF;
			IF (FBCalcPlungeGrindingMultiCycle.iStepSectionWork = 7) THEN
				(* Count the Plunge Cycle *)
				T_WorkTool.iTotalCountDownPlungeCycle:=T_WorkTool.iTotalCountDownPlungeCycle + 1;
			END_IF;
			IF (FBCalcPlungeGrindingMultiCycle.iStepSectionWork >= 1) AND (FBCalcPlungeGrindingMultiCycle.iStepSectionWork <= 6) THEN
			(* section 1 - 6 *)
				iTmpStartSection:=iStartSection + (FBCalcPlungeGrindingMultiCycle.iStepSectionWork - 1);
				rGrindFeederPlunge:=FBCalcPlungeGrindingMultiCycle.rGrindingRelativePosition;
				T_WorkTool.rGrindFeederPlunge:=rGrindFeederPlunge;
				T_WorkTool.rPitch:=T_Geometry.arSectionPitch[iTmpStartSection];
				T_WorkTool.rToolLength:=T_Geometry.arSectionLength[iTmpStartSection];
				FBToolCalcul(	xMicroRodActive:=xMicroRodActive,
								xBeckhoffDriveActive:=FALSE,
								T_WorkTool:= T_WorkTool);
				rTimeLeftWork:=rTimeLeftWork + T_WorkTool.rTimeLeftWork;
			END_IF;
			IF (FBCalcPlungeGrindingMultiCycle.iStepSectionWork = 0) THEN
				(* Calc Plunge *)
				IF T_AutoGeometryPara.xPlungeActivationGeometry THEN
					T_WorkTool.rPitch:=T_Geometry.arSectionPitch[iStartSection] * -1.0;
					T_WorkTool.rGrindFeederPlunge:=FBCalcPlungeGrindingMultiCycle.rGrindingRelativePosition;
					rToolFeedLength:=T_AutoGeometryPara.rPlungeLengthToolFeedGeometry;
					T_WorkTool.rToolLength:=rToolFeedLength;
					T_WorkTool.rToolRotationSpeed:=T_AutoGeometryPara.rSpeedToolRotationGeometry;
					FBToolCalcul(	xMicroRodActive:=xMicroRodActive,
									xBeckhoffDriveActive:=FALSE,
									T_WorkTool:= T_WorkTool);
					rSpeedToolFeed:=T_WorkTool.rToolFeederSpeedUnit * -1.0;
					IF (rSpeedToolFeed <> 0) THEN
						rTimeLeftWork:=rTimeLeftWork + T_WorkTool.rToolLength/rSpeedToolFeed;
					END_IF;
				ELSE
					(* No Plunging activation, than also is the GrindFeeder the master *)
					rPlungeGrind:=ABS(FBCalcPlungeGrindingMultiCycle.rGrindingRelativePosition);
					IF (T_AutoGeometryPara.rPlungeSpeedGrindFeedGeometry <> 0) THEN
						rTimeLeftWork:=rTimeLeftWork + (rPlungeGrind / T_AutoGeometryPara.rPlungeSpeedGrindFeedGeometry);
					END_IF;
				END_IF;
			END_IF;
			IF (FBCalcPlungeGrindingMultiCycle.iStepSectionWork = 7) THEN
				(* Calc Displace *)
				IF T_AutoGeometryPara.xDisplaceActivationGeometry THEN
					T_WorkTool.rPitch:=T_Geometry.arSectionPitch[iEndSection] * -1.0;
					T_WorkTool.rGrindFeederPlunge:=FBCalcPlungeGrindingMultiCycle.rGrindingRelativePosition;
					rToolFeedLength:=T_AutoGeometryPara.rDisplaceLengthToolFeedGeometry;
					T_WorkTool.rToolLength:=rToolFeedLength;
					T_WorkTool.rToolRotationSpeed:=T_AutoGeometryPara.rSpeedToolRotationGeometry;
					FBToolCalcul(	xMicroRodActive:=xMicroRodActive,
									xBeckhoffDriveActive:=FALSE,
									T_WorkTool:= T_WorkTool);
					rSpeedToolFeed:=T_WorkTool.rToolFeederSpeedUnit * -1.0;
					IF (rSpeedToolFeed <> 0) THEN
						rTimeLeftWork:=rTimeLeftWork + T_WorkTool.rToolLength/rSpeedToolFeed;
					END_IF;
				ELSE
					(* No Displace activation, than also is the GrindFeeder the master *)
					rDisplaceGrind:=ABS(FBCalcPlungeGrindingMultiCycle.rGrindingRelativePosition);
					IF (T_AutoGeometryPara.rDisplaceSpeedGrindFeedGeometry <> 0) THEN
						rTimeLeftWork:=rTimeLeftWork + (rDisplaceGrind / T_AutoGeometryPara.rDisplaceSpeedGrindFeedGeometry);
					END_IF;
				END_IF;
			END_IF;
		END_WHILE;
		IF (T_AutoGeometryPara.iCycleGeometry > 1) THEN
			rTimeLeftWork:=rTimeLeftWork * INT_TO_REAL(T_AutoGeometryPara.iCycleGeometry);
		END_IF;
	END_IF;
(**************iAutoProcess 2 --> AutoGroove********************************************************************************************************************************************************************************************************)
	IF (iAutoProcess = 2) THEN
	(* calculate the time for the process AutoGeometry or AutoGroove *)
		T_WorkTool.iTotalCountDownPlungeCycle:=0;
		(* Check Start and End Section of the ToolGeometry *)
		FOR ii:=1 TO 6 DO
			IF T_Geometry.axActiveSection[ii] THEN
				IF (iStartSection = 0) THEN
					iStartSection:=ii;
				END_IF;
				iEndSection:=ii;
			END_IF;
		END_FOR;
(*
		xResetFB:=TRUE;
		(* reset first the FB for calculate the grinding plunge for each sections *)
		FBCalcPlungeGrinding(	rToolDiameter:= rToolDiameter,
								rToolDiameterWithOffset:=rToolDiameterWithOffset,
								xReset:= xResetFB);
		rPlungeCycleGrindFeedGeometry:=1.0;
*)
		xResetFB:=TRUE;
		(* reset first the FB for calculate the grinding plunge for each sections *)
		FBCalcPlungeGrindingMultiCycle(	rToolDiameter:= rToolDiameter,
										rToolDiameterWithOffset:=rToolDiameterWithOffset,
										xReset:= xResetFB,
										xInit:=xInitFB);
		xInitFB:=TRUE;
		FBCalcPlungeGrindingMultiCycle(	T_Geometry:= T_Geometry,
										T_AutoGeometryPara:= T_AutoGeometryPara,
										rToolDiameter:= rToolDiameter,
										rToolDiameterWithOffset:=rToolDiameterWithOffset,
										rPlungeCycleGrindFeedGeometry:=rPlungeCycleGrindFeedGeometry,
										iStartSection:= iStartSection,
										iEndSection:= iEndSection,
										xReset:= xResetFB,
										xInit:=xInitFB);
		rPlungeCycleGrindFeedGeometry:=1.0;
		IF (iAutoProcess = 2) OR NOT(xMicroRodActive) THEN
			rPlungeCycleGrindFeedGeometry:=rToolDiameter;		(* for the groove process or for the MicroWire is not possible to work in more cycle, because of that it will set the tooldiamter *)
		END_IF;
		T_WorkTool.rToolRotationSpeed:=rToolRotationSpeed;
		xCalculation:=TRUE;
		WHILE(xCalculation) DO
			(* calculate the grinding way of each section *)
			FBCalcPlungeGrindingMultiCycle(	T_Geometry:= T_Geometry,
											T_AutoGeometryPara:= T_AutoGeometryPara,
											rToolDiameter:= rToolDiameter,
											rToolDiameterWithOffset:=rToolDiameterWithOffset,
											rPlungeCycleGrindFeedGeometry:=rPlungeCycleGrindFeedGeometry,
											iStartSection:= iStartSection,
											iEndSection:= iEndSection,
											xReset:= xResetFB,
											xInit:=xInitFB);
			IF FBCalcPlungeGrindingMultiCycle.xEndWorking THEN		(* check if the end of the to work Tool is reached *)
				xCalculation:=FALSE;
				EXIT;
			END_IF;
			IF (T_WorkTool.iTotalCountDownPlungeCycle >= 20) THEN	(* not possible to work a Tool in more that 20 cycle *)
				xCalculation:=FALSE;
				EXIT;
			END_IF;
			IF (FBCalcPlungeGrindingMultiCycle.iStepSectionWork = 7) THEN
				(* Count the Plunge Cycle *)
				T_WorkTool.iTotalCountDownPlungeCycle:=T_WorkTool.iTotalCountDownPlungeCycle + 1;
			END_IF;
			IF (FBCalcPlungeGrindingMultiCycle.iStepSectionWork >= 1) AND (FBCalcPlungeGrindingMultiCycle.iStepSectionWork <= 6) THEN
			(* section 1 - 6 *)
				iTmpStartSection:=iStartSection + (FBCalcPlungeGrindingMultiCycle.iStepSectionWork - 1);
				rGrindFeederPlunge:=FBCalcPlungeGrindingMultiCycle.rGrindingRelativePosition;
				T_WorkTool.rGrindFeederPlunge:=rGrindFeederPlunge;
				T_WorkTool.rPitch:=T_AutoGroovePara.rPitchGroove;
				T_WorkTool.rToolLength:=T_Geometry.arSectionLength[iTmpStartSection];
				FBToolCalcul(	xMicroRodActive:=xMicroRodActive,
								xBeckhoffDriveActive:=FALSE,
								T_WorkTool:= T_WorkTool);
				rTimeLeftWork:=rTimeLeftWork + T_WorkTool.rTimeLeftWork;
			END_IF;
			IF (FBCalcPlungeGrindingMultiCycle.iStepSectionWork = 0) THEN
				(* Calc Plunge *)
				IF T_AutoGroovePara.xPlungeActivationGroove  THEN
					T_WorkTool.rPitch:=T_AutoGroovePara.rPitchGroove * -1.0;
					T_WorkTool.rGrindFeederPlunge:=FBCalcPlungeGrindingMultiCycle.rGrindingRelativePosition;
					rToolFeedLength:=T_AutoGroovePara.rPlungeLengthToolFeedGroove;
					T_WorkTool.rToolLength:=rToolFeedLength;
					T_WorkTool.rToolRotationSpeed:=T_AutoGroovePara.rSpeedToolRotationGroove;
					FBToolCalcul(	xMicroRodActive:=xMicroRodActive,
									xBeckhoffDriveActive:=FALSE,
									T_WorkTool:= T_WorkTool);
					rSpeedToolFeed:=T_WorkTool.rToolFeederSpeedUnit * -1.0;
					IF (rSpeedToolFeed <> 0) THEN
						rTimeLeftWork:=rTimeLeftWork + T_WorkTool.rToolLength/rSpeedToolFeed;
					END_IF;
				ELSE
					(* No Plunging activation, than also is the GrindFeeder the master *)
					rPlungeGrind:=ABS(FBCalcPlungeGrindingMultiCycle.rGrindingRelativePosition);
					IF (T_AutoGroovePara.rPlungeSpeedGrindFeedGroove <> 0) THEN
						rTimeLeftWork:=rTimeLeftWork + (rPlungeGrind / T_AutoGroovePara.rPlungeSpeedGrindFeedGroove);
					END_IF;
				END_IF;
			END_IF;
			IF (FBCalcPlungeGrindingMultiCycle.iStepSectionWork = 7) THEN
				(* Calc Displace *)
				IF T_AutoGroovePara.xDisplaceActivationGroove  THEN
					T_WorkTool.rPitch:=T_AutoGroovePara.rPitchGroove * -1.0;
					T_WorkTool.rGrindFeederPlunge:=FBCalcPlungeGrindingMultiCycle.rGrindingRelativePosition;
					rToolFeedLength:=T_AutoGroovePara.rDisplaceLengthToolFeedGroove;
					T_WorkTool.rToolLength:=rToolFeedLength;
					T_WorkTool.rToolRotationSpeed:=T_AutoGroovePara.rSpeedToolRotationGroove;
					FBToolCalcul(	xMicroRodActive:=xMicroRodActive,
									xBeckhoffDriveActive:=FALSE,
									T_WorkTool:= T_WorkTool);
					rSpeedToolFeed:=T_WorkTool.rToolFeederSpeedUnit * -1.0;
					IF (rSpeedToolFeed <> 0) THEN
						rTimeLeftWork:=rTimeLeftWork + T_WorkTool.rToolLength/rSpeedToolFeed;
					END_IF;
				ELSE
					(* No Displace activation, than also is the GrindFeeder the master *)
					rDisplaceGrind:=ABS(FBCalcPlungeGrindingMultiCycle.rGrindingRelativePosition);
					IF (T_AutoGroovePara.rDisplaceSpeedGrindFeedGroove <> 0) THEN
						rTimeLeftWork:=rTimeLeftWork + (rPlungeGrind / T_AutoGroovePara.rDisplaceSpeedGrindFeedGroove);
					END_IF;
				END_IF;
			END_IF;
		END_WHILE;
		IF (T_AutoGroovePara.iNumberOfGrooves > 1) THEN
			rTimeLeftWork:=rTimeLeftWork * INT_TO_REAL(T_AutoGroovePara.iNumberOfGrooves);
			(* Berechnung zusätzlicher Weg und Zeit für Ausstechen & Einstechen ab 2. Zyklus*)
			rPlungeGrind:=ABS(T_ProcessPara.rSecurityPosGrindFeedProcess - T_ProcessPara.rToolDiameterProcess) * 2.0;
			rTimeAddLeftWorkPlungeGrind:= rPlungeGrind / T_ProcessPara.rSpeedForwardFastGrindFeed;
			(* Berechnung zusätzlicher Weg und Zeit  Ausstechen für letzten Zyklus*)
			rPlungeGrind2:=ABS(T_ProcessPara.rSecurityPosGrindFeedProcess - T_ProcessPara.rToolDiameterProcess);
			rTimeAddLeftWorkPlungeGrind2:= rPlungeGrind2 / T_ProcessPara.rSpeedForwardFastGrindFeed;
			(*Berechnung zusätzlicher Weg und Zeit  Rückfahren  ab 2. Zyklus*)
			rToolLength:=0;
			FOR ii:=1 TO 6 DO
				IF T_Geometry.axActiveSection[ii] THEN
					rToolLength:=rToolLength + T_Geometry.arSectionLength[ii];
				END_IF;
			END_FOR;
			rTimeAddLeftWorkToolFeed:= rToolLength*10/T_ProcessPara.rSpeedStartPosToolFeedProcess;
			(*Berchnung der gesamten zusätzlichen Prozesszeit*)
			rTimeAddLeftWork:=(rTimeAddLeftWorkPlungeGrind + rTimeAddLeftWorkToolFeed) * (T_AutoGroovePara.iNumberOfGrooves -1);
			rTimeAddLeftWork:= rTimeAddLeftWork+rTimeAddLeftWorkPlungeGrind2;
			rTimeLeftWork:=rTimeLeftWork + rTimeAddLeftWork;
		END_IF;
	END_IF;
(**************iAutoProcess 0***********************************************************************************************************************************************************************************************************************)
	IF (iAutoProcess = 0) THEN
	(* Calculate the time for the process ToolCalibration *)
		T_WorkTool.rToolRotationSpeed:=T_CalibrationPara.rSpeedToolRotationCalib;
		T_WorkTool.rGrindFeederPlunge:=T_ProcessPara.rOffsetBeforeToolDiaGrindFeedProcess;
		T_WorkTool.rPitch:=T_CalibrationPara.rPitchCalib;
		T_WorkTool.rToolLength:=T_CalibrationPara.rToolLengthCylinderPartCalib;
		FBToolCalcul(	xMicroRodActive:=xMicroRodActive,
						xBeckhoffDriveActive:=FALSE,
						T_WorkTool:= T_WorkTool);
		rTimeLeftWork:=rTimeLeftWork + T_WorkTool.rTimeLeftWork;
		IF T_CalibrationPara.xPlungeActivationCalib THEN
			T_WorkTool.rPitch:=T_CalibrationPara.rPitchCalib;
			T_WorkTool.rGrindFeederPlunge:=T_ProcessPara.rOffsetBeforeToolDiaGrindFeedProcess;
			rToolFeedLength:=T_CalibrationPara.rPlungeLengthToolFeedCalib;
			T_WorkTool.rToolLength:=rToolFeedLength;
			FBToolCalcul(	xMicroRodActive:=xMicroRodActive,
							xBeckhoffDriveActive:=FALSE,
							T_WorkTool:= T_WorkTool);
			rSpeedToolFeed:=T_WorkTool.rToolFeederSpeedUnit;
			IF (rSpeedToolFeed <> 0) THEN
				rTimeLeftWork:=rTimeLeftWork + T_WorkTool.rToolLength/ABS(rSpeedToolFeed);
			END_IF;
		ELSE
			(* No Plunging activation, than also is the GrindFeeder the master *)
			rPlungeGrind:=T_ProcessPara.rOffsetBeforeToolDiaGrindFeedProcess;
			rTimeLeftWork:=rTimeLeftWork + (rPlungeGrind / T_CalibrationPara.rPlungeSpeedGrindFeedCalib);
		END_IF;


		IF T_CalibrationPara.xDisplaceActivationCalib THEN
			T_WorkTool.rPitch:=T_CalibrationPara.rPitchCalib * -1.0;
			T_WorkTool.rGrindFeederPlunge:=T_ProcessPara.rOffsetBeforeToolDiaGrindFeedProcess;
			rToolFeedLength:=T_CalibrationPara.rDisplaceLengthToolFeedCalib;
			T_WorkTool.rToolLength:=rToolFeedLength;
			FBToolCalcul(	xMicroRodActive:=xMicroRodActive,
							xBeckhoffDriveActive:=FALSE,
							T_WorkTool:= T_WorkTool);
			rSpeedToolFeed:=T_WorkTool.rToolFeederSpeedUnit;
			IF (rSpeedToolFeed <> 0) THEN
				rTimeLeftWork:=rTimeLeftWork + T_WorkTool.rToolLength/ABS(rSpeedToolFeed);
			END_IF;
		ELSE
			(* No Displace activation, than also is the GrindFeeder the master *)
			rDisplaceGrind:=T_ProcessPara.rOffsetBeforeToolDiaGrindFeedProcess;
			rTimeLeftWork:=rTimeLeftWork + (rDisplaceGrind / T_CalibrationPara.rDisplaceSpeedGrindFeedCalib);
		END_IF;
	END_IF;
	rProcessTime:=rTimeLeftWork;
END_FUNCTION_BLOCK

(* POU GENERAL/FB_TOOL_CALCUL, ST *)
FUNCTION_BLOCK FB_TOOL_CALCUL
VAR_INPUT
	xMicroRodActive: BOOL;			(* choice of the machine MicroWire or MicroRod *)
	xBeckhoffDriveActive: BOOL;		(* choice of the Axis Beckhoff or EcoStep *)
END_VAR
VAR_IN_OUT
	T_WorkTool:ST_WORKTOOL;		(* Tool Parameter *)
END_VAR
VAR_OUTPUT
END_VAR
VAR
END_VAR
(****************************************************************************************************************************************************)
(***********                                  This Functionblock calculate all needed parameter for work a Tool                                            ************)
(****************************************************************************************************************************************************)
(* calcul ToolRotation Speed in inc/64s *)
	IF (T_WorkTool.rToolRotationSpeed <> 0) AND (T_WorkTool.rToolRightGearRatio <> 0) THEN
		T_WorkTool.rToolRotationSpeedMotor:=((T_WorkTool.rToolRotationSpeed / 60.0) * 8000.0 * 64.0) / T_WorkTool.rToolRightGearRatio;
	ELSE
		RETURN;	(* Exit FB *)
	END_IF;
(* calcul ToolFeeder Speed in mm/s *)
	T_WorkTool.rToolFeederSpeedUnit:=T_WorkTool.rPitch * (T_WorkTool.rToolRotationSpeed / 60.0);
(* calcul ToolFeeder Speed in inc/64s Relativ *)
	T_WorkTool.rToolFeederSpeedMotorRel:=T_WorkTool.rToolFeederScaleFactor * T_WorkTool.rToolFeederSpeedUnit * 64.0;
(* calcul ToolFeeder Speed in inc/64s Relativ *)
	T_WorkTool.rToolFeederSpeedMotorAbs:=(T_WorkTool.rToolRotationSpeedMotor * T_WorkTool.rToolRightGearRatio) + T_WorkTool.rToolFeederSpeedMotorRel;
(* Set ToolFeeder GearDivider *)
	T_WorkTool.iToolFeederGearDivider:=T_WorkTool.iBaseGearDivider;
	IF xMicroRodActive THEN
	(* calcul ToolFeeder GearFactor *)
		IF (T_WorkTool.rPitch <> 0) THEN
			T_WorkTool.iToolFeederGearFactor:=REAL_TO_INT(INT_TO_REAL(T_WorkTool.iBaseGearDivider) / (T_WorkTool.rToolRotationSpeedMotor / T_WorkTool.rToolFeederSpeedMotorRel));
		ELSE
			T_WorkTool.iToolFeederGearFactor:=REAL_TO_INT(INT_TO_REAL(T_WorkTool.iToolFeederGearDivider) * T_WorkTool.rToolRightGearRatio);
		END_IF;
	ELSE
	(* calcul ToolFeeder GearFactor *)
		IF (T_WorkTool.rPitch <> 0) THEN
			T_WorkTool.iToolFeederGearFactor:=REAL_TO_INT(INT_TO_REAL(T_WorkTool.iBaseGearDivider) / (T_WorkTool.rToolRotationSpeedMotor / T_WorkTool.rToolFeederSpeedMotorAbs));
		ELSE
			T_WorkTool.iToolFeederGearFactor:=REAL_TO_INT(INT_TO_REAL(T_WorkTool.iToolFeederGearDivider) * T_WorkTool.rToolRightGearRatio);
		END_IF;
	END_IF;
(* calcul Time to work *)
	IF (T_WorkTool.rToolFeederSpeedUnit <> 0) THEN
		T_WorkTool.rTimeLeftWork:=(T_WorkTool.rToolLength * 10.0) / ABS(T_WorkTool.rToolFeederSpeedUnit);
	ELSE
		T_WorkTool.rTimeLeftWork:=0.0;
	END_IF;
(* calcul ToolFeeder relative Position to drive *)
	T_WorkTool.rToolFeederRelPositionUnit:=T_WorkTool.rToolLength * 10.0;
	T_WorkTool.rToolFeederRelPositionMotor:=T_WorkTool.rToolFeederRelPositionUnit * T_WorkTool.rToolFeederScaleFactor;
(* calcul GrindFeeder Speed in um/s *)
	IF (T_WorkTool.rTimeLeftWork <> 0) THEN
		T_WorkTool.rGrindFeederSpeedUnit:=T_WorkTool.rGrindFeederPlunge / T_WorkTool.rTimeLeftWork;
	ELSE
		T_WorkTool.rGrindFeederSpeedUnit:=0.0;
	END_IF;
(* calcul GrindFeeder Speed in inc/s *)
	T_WorkTool.rGrindFeederSpeedMotor:=T_WorkTool.rGrindFeederSpeedUnit * T_WorkTool.rGrindFeederScaleFactor * 64.0;
END_FUNCTION_BLOCK

(* POU GENERAL/FB_CALC_PLUNGE_GRINDING, ST *)
FUNCTION_BLOCK FB_CALC_PLUNGE_GRINDING
VAR_INPUT
	T_Geometry:ST_GEOMETRY;								(* Structure of the NovRAM parameter *)
	T_AutoGeometryPara:ST_EXCHG_PARAM_AUTOGEOMETRY;	(* Structure of the NovRAM parameter *)
	rToolDiameter:REAL;					(* diameter of the unworked Tool *)
	rToolDiameterWithOffset:REAL;			(* diameter of the unworked Tool plus the offset for plunge and displace procedure *)
	rPlungeCycleGrindFeedGeometry:REAL;	(* max grinding plunging per cycle *)
	iStartSection:INT;						(* number of the start section *)
	iEndSection:INT;						(* number of the end section *)
END_VAR
VAR_IN_OUT
	xReset:BOOL;						(* resetting of the FB *)
END_VAR
VAR_OUTPUT
	iStepSectionWork:INT;				(* actual worked section number *)
	rGrindingRelativePosition:REAL;		(* relative way of the GrindFeeder plunge *)
	xEndWorking:BOOL;				(* end of the hole working procedure *)
	xError:BOOL;						(* error flag *)
END_VAR
VAR
(***S***)
	rActualPositionGrindFeedStart: ARRAY [0..7] OF REAL;	(* 0=StartPos Plunge,1-6=Dynamic StartPos Section 1-6, 7=StartPos Displace *)
	rActualPositionGrindFeedEnd: ARRAY [0..7] OF REAL;	(* 0=EndPos Plunge,1-6=Dynamic EndPos Section 1-6, 7=EndPos Displace *)
	rDistanceToWorkedTool: REAL;
	ii: INT;
	iStepSection: INT;
	axWorkEndSection: ARRAY [0..7] OF BOOL;
	xCheckEnd: BOOL;
	rTmpActualPositionGrindFeedStart:REAL;
	iStepCheckSection: INT;
	rTmpDistance: REAL;
	rGrinded: REAL;
END_VAR
(****************************************************************************************************************************************************)
(***********      This Functionblock calculate the plunge way for the GrindFeeder axis for the geometry sections  1-6        ************)
(***********                                           It calculate also the plunge and displace procedure							    ************)
(****************************************************************************************************************************************************)
IF xReset THEN
	xReset:=FALSE;
	iStepSection:=0;
	FOR ii:=0 TO 7 DO
		rActualPositionGrindFeedStart[ii]:=rToolDiameterWithOffset;
		rActualPositionGrindFeedEnd[ii]:=rToolDiameterWithOffset;
		axWorkEndSection[ii]:=FALSE;
	END_FOR;
	rActualPositionGrindFeedStart[0]:=rToolDiameterWithOffset;
	rActualPositionGrindFeedEnd[7]:=rToolDiameterWithOffset;
	rTmpActualPositionGrindFeedStart:=rToolDiameterWithOffset;
	rGrindingRelativePosition:=0.0;
	iStepSectionWork:=0;
	RETURN;
END_IF;
xError:=FALSE;
(* check the settled start and end section *)
IF (iStartSection < 1) OR (iStartSection > 6) THEN
	xError:=TRUE;
	RETURN;
END_IF;
IF (iEndSection < 1) OR (iEndSection > 6) THEN
	xError:=TRUE;
	RETURN;
END_IF;
IF (iStepSection < 0) OR (iStepSection > 7) THEN
	xError:=TRUE;
	RETURN;
END_IF;

CASE iStepSection OF
	(* plunge procedure *)
		0:	iStepCheckSection:=1;
			xCheckEnd:=TRUE;
			(* Check if the end of all section is reached *)
			FOR ii:=iStartSection TO iEndSection DO
				IF (rActualPositionGrindFeedStart[iStepCheckSection] <> T_Geometry.arStartDiameter[ii]) THEN
					xCheckEnd:=FALSE;
				END_IF;
				IF (rActualPositionGrindFeedEnd[iStepCheckSection] <> T_Geometry.arEndDiameter[ii]) THEN
					xCheckEnd:=FALSE;
				END_IF;
				iStepCheckSection:=iStepCheckSection + 1;
			END_FOR;
			xEndWorking:=xCheckEnd;
			IF xEndWorking THEN
				rGrindingRelativePosition:=0.0;
				RETURN;
			END_IF;
			IF (T_Geometry.arStartDiameter[iStartSection] = rActualPositionGrindFeedEnd[0]) THEN	(* check if the defined ToolDiameter for the plunge procedure is reached *)
				axWorkEndSection[0]:=TRUE;
				rGrindingRelativePosition:=rToolDiameterWithOffset - T_Geometry.arStartDiameter[iStartSection];
			END_IF;
			IF NOT(axWorkEndSection[0]) THEN
			(* if the end of the plunge procedure is not reached, then calculate the plunge way of the plunge procedure *)
				rGrindingRelativePosition:=(rToolDiameterWithOffset - rActualPositionGrindFeedEnd[0]) + rPlungeCycleGrindFeedGeometry;
				IF ((rToolDiameterWithOffset - rGrindingRelativePosition) <= T_Geometry.arStartDiameter[iStartSection]) THEN
					rGrindingRelativePosition:=rToolDiameterWithOffset - T_Geometry.arStartDiameter[iStartSection];
				END_IF;
			END_IF;
			rActualPositionGrindFeedStart[0]:=rToolDiameterWithOffset;	(* the start zero section of the geometry is always the diameter of the Tool *)
			rActualPositionGrindFeedEnd[0]:=rToolDiameterWithOffset - rGrindingRelativePosition;	(* calcualte the plunge way *)
			iStepSectionWork:=iStepSection;	(* set the actual section which is working *)
			iStepSection:=iStepSection + 1;		(* go to the next section *)
	(* geometry section 1,2,3,4,5 and 6 *)
	1,2,3,4,5,6:	rGrinded:=(rActualPositionGrindFeedStart[iStepSection] - rActualPositionGrindFeedEnd[iStepSection - 1]);	(* calculate the difference of the worked section before to the unworked section after *)
			IF (rGrinded < 0) THEN
				rGrinded:=rGrinded;
			END_IF;
			rActualPositionGrindFeedStart[iStepSection]:=rActualPositionGrindFeedStart[iStepSection] - rGrinded;		(* set the new diameter of the section which will go to work *)
			rTmpDistance:=T_Geometry.arStartDiameter[iStartSection + (iStepSection - 1)] - T_Geometry.arEndDiameter[iStartSection + (iStepSection - 1)]; (* set the difference of the start and end diameter of the section *)
			IF (rActualPositionGrindFeedStart[iStepSection] < T_Geometry.arStartDiameter[iStartSection + (iStepSection - 1)]) THEN	(* correct of the to grind Tool diameter *)
				rActualPositionGrindFeedStart[iStepSection]:=T_Geometry.arStartDiameter[iStartSection + (iStepSection - 1)];
			END_IF;
			rGrindingRelativePosition:=rPlungeCycleGrindFeedGeometry - rGrinded;	(* calculate the effectiv way for the plunge *)
			IF (rGrinded >= rPlungeCycleGrindFeedGeometry) THEN				(* check if the to grinding way is grater than the defined max grinding *)
				IF (rActualPositionGrindFeedStart[iStepSection] < T_Geometry.arEndDiameter[iStartSection + (iStepSection - 1)]) THEN
				(* correct the effective way for the plunge, because it can not work more than the defined grinding way *)
					rGrindingRelativePosition:=rActualPositionGrindFeedStart[iStepSection] - T_Geometry.arEndDiameter[iStartSection + (iStepSection - 1)];
				END_IF;
			ELSE
				IF (rTmpDistance = 0) THEN
				(* a cylinder part will now work *)
					rGrindingRelativePosition:=0.0;
				ELSE
					(* a cone part will now work *)
					rTmpDistance:=T_Geometry.arStartDiameter[iStartSection + (iStepSection - 1)] - rActualPositionGrindFeedEnd[iStepSection];
					rGrindingRelativePosition:=rTmpDistance + rPlungeCycleGrindFeedGeometry;
					IF ((T_Geometry.arStartDiameter[iStartSection + (iStepSection - 1)] - rGrindingRelativePosition) < T_Geometry.arEndDiameter[iStartSection + (iStepSection - 1)]) THEN
					(* correct the effective way for the plunge, because it can not work more than the defined grinding way *)
						rGrindingRelativePosition:=T_Geometry.arStartDiameter[iStartSection + (iStepSection - 1)] - T_Geometry.arEndDiameter[iStartSection + (iStepSection - 1)];
					END_IF;
				END_IF;
			END_IF;
			rActualPositionGrindFeedEnd[iStepSection]:=rActualPositionGrindFeedStart[iStepSection] - rGrindingRelativePosition;	(* calculate the end position of the section *)
			iStepSectionWork:=iStepSection;		(* set the actual section which is working *)
			IF ((iStepSection + (iStartSection - 1)) < iEndSection) THEN	(* check if the end section is active *)
				iStepSection:=iStepSection + 1;
			ELSE
				iStepSection:=7;	(* end section is reached-->go the displace procedure *)
			END_IF;
	(* plunge procedure *)
	7:		rActualPositionGrindFeedStart[7]:=rActualPositionGrindFeedEnd[iEndSection - (iStartSection - 1)];	(* set the new diameter of the section which will going to work *)
			rDistanceToWorkedTool:=rActualPositionGrindFeedStart[7] - rToolDiameterWithOffset;	(* check the distance to the end diameter, which will go to work *)
			rGrindingRelativePosition:=rDistanceToWorkedTool;
			IF (rActualPositionGrindFeedStart[5] = T_Geometry.arEndDiameter[iEndSection]) THEN
				axWorkEndSection[7]:=TRUE;		(* the end of this section is reached *)
			ELSE
				axWorkEndSection[7]:=FALSE;		(* the end of this section is reached *)
			END_IF;
			rActualPositionGrindFeedEnd[7]:=rToolDiameterWithOffset;
			iStepSectionWork:=iStepSection;		(* set the actual section which is working *)
			iStepSection:=0;
END_CASE;
END_FUNCTION_BLOCK

(* POU GENERAL/FB_CALC_PLUNGE_GRINDING_MultiCycle, ST *)
FUNCTION_BLOCK FB_CALC_PLUNGE_GRINDING_MultiCycle
VAR_INPUT
	T_Geometry:ST_GEOMETRY;								(* Structure of the NovRAM parameter *)
	T_AutoGeometryPara:ST_EXCHG_PARAM_AUTOGEOMETRY;	(* Structure of the NovRAM parameter *)
	rToolDiameter:REAL;					(* diameter of the unworked Tool *)
	rToolDiameterWithOffset:REAL;			(* diameter of the unworked Tool plus the offset for plunge and displace procedure *)
	rPlungeCycleGrindFeedGeometry:REAL;	(* max grinding plunging per cycle *)
	iStartSection:INT;						(* number of the start section *)
	iEndSection:INT;						(* number of the end section *)
END_VAR
VAR_IN_OUT
	xReset:BOOL;						(* resetting of the FB *)
	xInit:BOOL;							(* Init of the FB *)
END_VAR
VAR_OUTPUT
	iStepSectionWork:INT;				(* actual worked section number *)
	rGrindingRelativePosition:REAL;		(* relative way of the GrindFeeder plunge *)
	xEndWorking:BOOL;				(* end of the hole working procedure *)
	xError:BOOL;						(* error flag *)
END_VAR
VAR
	rActualPositionGrindFeedStart: ARRAY [0..7] OF REAL;	(* 0=StartPos Plunge,1-4=Dynamic StartPos Section 1-4, 5=StartPos Displace *)
	rActualPositionGrindFeedEnd: ARRAY [0..7] OF REAL;	(* 0=EndPos Plunge,1-4=Dynamic EndPos Section 1-4, 5=EndPos Displace *)
	rDistanceToWorkedTool: REAL;
	ii: INT;
	iStepSection: INT;
	axWorkEndSection: ARRAY [0..7] OF BOOL;
	xCheckEnd: BOOL;
	rTmpActualPositionGrindFeedStart:REAL;
	iStepCheckSection: INT;
	rTmpDistance: REAL;
	rGrinded: REAL;
	rMaxPlungeWay:REAL;
	rMaxPlungeWayStepOffset:REAL;
        	diNrOfAdditionalPlungeCycle:DINT;
END_VAR
(*****************************************************************************************************************************************************)
(***********      This Functionblock calculates the plunge way for the GrindFeeder axis for the geometry sections  1-6        ************)
(***********                                           It calculates also the plunge and displace procedure							    *************)
(*****************************************************************************************************************************************************)
IF xReset THEN
	xReset:=FALSE;
	iStepSection:=0;
	FOR ii:=0 TO 7 DO
		rActualPositionGrindFeedStart[ii]:=rToolDiameterWithOffset;
		rActualPositionGrindFeedEnd[ii]:=rToolDiameterWithOffset;
		axWorkEndSection[ii]:=FALSE;
	END_FOR;
	rActualPositionGrindFeedStart[0]:=rToolDiameterWithOffset;
	rActualPositionGrindFeedEnd[7]:=rToolDiameterWithOffset;
	rTmpActualPositionGrindFeedStart:=rToolDiameterWithOffset;
	rGrindingRelativePosition:=0.0;
	iStepSectionWork:=0;
	rMaxPlungeWay:=0.0;
	RETURN;
END_IF;
(*22.12.2009: KFS 	{   *)
IF xInit THEN
	xInit:=FALSE;
(*	rMaxPlungeWay:= rToolDiameter - T_Geometry.arEndDiameter[iEndSection]; (*Calculation of the max. plunge way*)*)
	rMaxPlungeWay:= rToolDiameterWithOffset - T_Geometry.arEndDiameter[iEndSection]; (*Calculation of the max. plunge way*)
	diNrOfAdditionalPlungeCycle:= MODTURNS (rMaxPlungeWay, rPlungeCycleGrindFeedGeometry);
	IF diNrOfAdditionalPlungeCycle > 0 THEN
		rMaxPlungeWayStepOffset:=LMOD(rMaxPlungeWay, rPlungeCycleGrindFeedGeometry);
		IF rMaxPlungeWayStepOffset > 0 THEN
			diNrOfAdditionalPlungeCycle:=diNrOfAdditionalPlungeCycle + 1;
		END_IF;
		rMaxPlungeWay:= rPlungeCycleGrindFeedGeometry * diNrOfAdditionalPlungeCycle;
	END_IF;
	iStepCheckSection:=1;
	(*Add the max plunge way on all start- and stop- points of the geometry*)
	FOR ii:=iStartSection TO iEndSection DO
(*		rActualPositionGrindFeedStart[iStepCheckSection] := rToolDiameterWithOffset - rToolDiameter +T_Geometry.arStartDiameter[ii] + rMaxPlungeWay;
		rActualPositionGrindFeedEnd[iStepCheckSection]:= rToolDiameterWithOffset  - rToolDiameter + T_Geometry.arEndDiameter[ii]+ rMaxPlungeWay; *)
		rActualPositionGrindFeedStart[iStepCheckSection] := T_Geometry.arStartDiameter[ii] + rMaxPlungeWay;
		rActualPositionGrindFeedEnd[iStepCheckSection]:=  T_Geometry.arEndDiameter[ii]+ rMaxPlungeWay;
		iStepCheckSection:=iStepCheckSection + 1;
	END_FOR;
	rActualPositionGrindFeedStart[0]:=rActualPositionGrindFeedStart[1];
	rActualPositionGrindFeedEnd[0]:=rActualPositionGrindFeedStart[1];
	RETURN;
END_IF;
(*22.12.2009: KFS 	}   *)
xError:=FALSE;
(* check the settled start and end section *)
IF (iStartSection < 1) OR (iStartSection > 6) THEN
	xError:=TRUE;
	RETURN;
END_IF;
IF (iEndSection < 1) OR (iEndSection > 6) THEN
	xError:=TRUE;
	RETURN;
END_IF;
IF (iStepSection < 0) OR (iStepSection > 7) THEN
	xError:=TRUE;
	RETURN;
END_IF;
CASE iStepSection OF
	(* plunge procedure *)
		0:	iStepCheckSection:=1;
			xCheckEnd:=TRUE;
			(* Check if the end of all section is reached *)
			FOR ii:=iStartSection TO iEndSection DO
				IF (rActualPositionGrindFeedStart[iStepCheckSection] <> T_Geometry.arStartDiameter[ii]) THEN
					xCheckEnd:=FALSE;
				END_IF;
				IF (rActualPositionGrindFeedEnd[iStepCheckSection] <> T_Geometry.arEndDiameter[ii]) THEN
					xCheckEnd:=FALSE;
				END_IF;
				iStepCheckSection:=iStepCheckSection + 1;
			END_FOR;
			xEndWorking:=xCheckEnd;
			IF xEndWorking THEN
				rGrindingRelativePosition:=0.0;
				RETURN;
			END_IF;
			IF (T_Geometry.arStartDiameter[iStartSection] = rActualPositionGrindFeedEnd[0]) THEN	(* check if the defined ToolDiameter for the plunge procedure is reached *)
				axWorkEndSection[0]:=TRUE;
				rGrindingRelativePosition:=rToolDiameterWithOffset - T_Geometry.arStartDiameter[iStartSection];
			END_IF;
			IF NOT(axWorkEndSection[0]) THEN
			(* if the end of the plunge procedure is not reached, then calculate the plunge way of the plunge procedure *)
				rGrindingRelativePosition:=(rToolDiameterWithOffset - rActualPositionGrindFeedEnd[0]) + rPlungeCycleGrindFeedGeometry;
				IF ((rToolDiameterWithOffset - rGrindingRelativePosition) <= T_Geometry.arStartDiameter[iStartSection]) THEN
					rGrindingRelativePosition:=rToolDiameterWithOffset - T_Geometry.arStartDiameter[iStartSection];
				END_IF;
			END_IF;
			(*22.12.2009: KFS 	{   *)
			(*
			rActualPositionGrindFeedStart[0]:=rToolDiameterWithOffset;	(* the start zero section of the geometry is always the diameter of the Tool *)
			*)
			rActualPositionGrindFeedStart[0]:=rToolDiameterWithOffset - rGrindingRelativePosition;	(* the start zero section of the geometry is always the diameter of the Tool *)
			(*22.12.2009: KFS 	}   *)
			rActualPositionGrindFeedEnd[0]:=rToolDiameterWithOffset - rGrindingRelativePosition;	(* calcualte the plunge way *)
			iStepSectionWork:=iStepSection;	(* set the actual section which is working *)
			iStepSection:=iStepSection + 1;		(* go to the next section *)
	(* geometry section 1,2,3, 4,5 and 6 *)
	1..6:	rGrinded:=(rActualPositionGrindFeedStart[iStepSection] - rActualPositionGrindFeedEnd[iStepSection - 1]);	(* calculate the difference of the worked section before to the unworked section after *)
			IF (rGrinded < 0) THEN
				rGrinded:=rGrinded;
			END_IF;
			rActualPositionGrindFeedStart[iStepSection]:=rActualPositionGrindFeedStart[iStepSection] - rGrinded;		(* set the new diameter of the section which will going to work *)
			rTmpDistance:=T_Geometry.arStartDiameter[iStartSection + (iStepSection - 1)] - T_Geometry.arEndDiameter[iStartSection + (iStepSection - 1)]; (* set the difference of the start and end diameter of the section *)
			IF (rActualPositionGrindFeedStart[iStepSection] < T_Geometry.arStartDiameter[iStartSection + (iStepSection - 1)]) THEN	(* correct of the to grind Tool diameter *)
				rActualPositionGrindFeedStart[iStepSection]:=T_Geometry.arStartDiameter[iStartSection + (iStepSection - 1)];
			END_IF;
			rGrindingRelativePosition:=rPlungeCycleGrindFeedGeometry - rGrinded ;	(* calculate the effectiv way for the plunge *)
(*			IF (rGrinded >= rPlungeCycleGrindFeedGeometry) THEN				(* check if the to grinding way is grater than the defined max grinding *) *)
			IF (rGrinded > rPlungeCycleGrindFeedGeometry) THEN				(* check if the to grinding way is grater than the defined max grinding *)
				IF (rActualPositionGrindFeedStart[iStepSection] < T_Geometry.arEndDiameter[iStartSection + (iStepSection - 1)]) THEN
				(* correct the effective way for the plunge, because it can not work more than the defined grinding way *)
					rGrindingRelativePosition:=rActualPositionGrindFeedStart[iStepSection] - T_Geometry.arEndDiameter[iStartSection + (iStepSection - 1)];
				END_IF;
			ELSE
				IF (rTmpDistance = 0) THEN
				(* a cylinder part will now work *)
					rGrindingRelativePosition:=0.0;
				ELSE
					(* a cone part will now work *)
					rGrindingRelativePosition:=rTmpDistance;
					IF ((T_Geometry.arStartDiameter[iStartSection + (iStepSection - 1)] - rGrindingRelativePosition) < T_Geometry.arEndDiameter[iStartSection + (iStepSection - 1)]) THEN
					(* correct the effective way for the plunge, because it can not work more than the defined grinding way *)
						rGrindingRelativePosition:=T_Geometry.arStartDiameter[iStartSection + (iStepSection - 1)] - T_Geometry.arEndDiameter[iStartSection + (iStepSection - 1)];
					END_IF;
				END_IF;
			END_IF;
			rActualPositionGrindFeedEnd[iStepSection]:=rActualPositionGrindFeedStart[iStepSection] - rGrindingRelativePosition;	(* calculate the end position of the section *)

			iStepSectionWork:=iStepSection;		(* set the actual section which is working *)
			IF ((iStepSection + (iStartSection - 1)) < iEndSection) THEN	(* check if the end section is active *)
				iStepSection:=iStepSection + 1;
			ELSE
				iStepSection:=7;	(* end section is reached-->go the displace procedure *)
			END_IF;
	(* plunge procedure *)
	7:		rActualPositionGrindFeedStart[7]:=rActualPositionGrindFeedEnd[iEndSection - (iStartSection - 1)];	(* set the new diameter of the section which will going to work *)
			rDistanceToWorkedTool:=rActualPositionGrindFeedStart[7] - rToolDiameterWithOffset;	(* check the distance to the end diameter, which will go to work *)
			rGrindingRelativePosition:=rDistanceToWorkedTool;
			IF (rActualPositionGrindFeedStart[7] = T_Geometry.arEndDiameter[iEndSection]) THEN
				axWorkEndSection[7]:=TRUE;		(* the end of this section is reached *)
			ELSE
				axWorkEndSection[7]:=FALSE;		(* the end of this section is not reached *)
			END_IF;
			rActualPositionGrindFeedEnd[7]:=rToolDiameterWithOffset;
			iStepSectionWork:=iStepSection;		(* set the actual section which is working *)
			iStepSection:=0;
END_CASE;
END_FUNCTION_BLOCK

(* POU PRG_VISU_LAYER5/FB_VISU/iFctGetEditParaList, ST *)
FUNCTION iFctGetEditParaList : INT
VAR_INPUT
	dwActualPage:DWORD;		(* activate page on the visualisation *)
	xMicroRodActive: BOOL;		(* choice of the machine MicroWire or MicroRod *)
	iSelectParaList:INT;			(* parameter list choiced on the QVis *)
	iSelectParaListTeachRot:INT;	(* parameter list choiced on the QVis for teach ToolRotation *)
END_VAR
VAR
	iTmpRetEditParaList: INT;
END_VAR
(****************************************************************************************************************************************************)
(***********          This Function check the state of the parameter level and give the number of the parameter list                ************)
(****************************************************************************************************************************************************)
iTmpRetEditParaList:=0;
CASE dwActualPage OF
	110:	IF xMicroRodActive THEN
			iTmpRetEditParaList:=111;
		ELSE
			iTmpRetEditParaList:=110;
		END_IF;
	120:	IF (iSelectParaList = 0) OR (iSelectParaList = 1) THEN
			IF xMicroRodActive THEN
				iTmpRetEditParaList:=123;
			ELSE
				iTmpRetEditParaList:=120;
			END_IF;
		END_IF;
		IF (iSelectParaList = 2) THEN
			iTmpRetEditParaList:=121;
		END_IF;
		IF (iSelectParaList = 3) THEN
			IF xMicroRodActive THEN
				iTmpRetEditParaList:=125;
			ELSE
				iTmpRetEditParaList:=122;
			END_IF;
		END_IF;
	130:	IF xMicroRodActive THEN
			iTmpRetEditParaList:=131;
		ELSE
			iTmpRetEditParaList:=130;
		END_IF;
	140:	iTmpRetEditParaList:=140;
	150:	iTmpRetEditParaList:=150;
	210:	IF (iSelectParaListTeachRot = 0) OR (iSelectParaListTeachRot = 1) THEN
			iTmpRetEditParaList:=210;
		END_IF;
		IF (iSelectParaListTeachRot = 2) THEN
			iTmpRetEditParaList:=211;
		END_IF;
		IF (iSelectParaListTeachRot = 3) THEN
			iTmpRetEditParaList:=212;
		END_IF;
	220:	iTmpRetEditParaList:=0;
	230:	iTmpRetEditParaList:=230;
	310:IF xMicroRodActive THEN
			iTmpRetEditParaList:=311;
		ELSE
			iTmpRetEditParaList:=310;
		END_IF;
	320:	iTmpRetEditParaList:=0;
	410:	iTmpRetEditParaList:=410;
	420:	iTmpRetEditParaList:=0;
	430:	iTmpRetEditParaList:=0;
END_CASE;
iFctGetEditParaList:=iTmpRetEditParaList;
END_FUNCTION

(* POU PRG_VISU_LAYER5/FB_VISU/iFctReturnConfMessage, ST *)
FUNCTION iFctReturnConfMessage : INT
VAR_INPUT
	iNumAction:INT;	(* number of called action on the visualisation *)
END_VAR
VAR
END_VAR
(****************************************************************************************************************************************************)
(***********                      This Function check the action on the visu and gives a correspond message number                     ************)
(****************************************************************************************************************************************************)
	CASE iNumAction OF
	(* Action exceeded Timeout *)
	-1:	iFctReturnConfMessage:=102;
	(* NovRAM, 'Parameter saved' with confirmation *)
	1005:	iFctReturnConfMessage:=1;
	(* NovRAM, 'Parameter saved' without confirmation *)
	1006:	iFctReturnConfMessage:=1;
	(* Reference machine done *)
	1110:	iFctReturnConfMessage:=23;
	(* Process machine done *)
	1150:	iFctReturnConfMessage:=21;
	(* Process station done *)
	1151..1153:	iFctReturnConfMessage:=22;
	(* change page, no message *)
	10001..10999:	iFctReturnConfMessage:=0;
	(* Info , 'Confirm action' *)
	ELSE	iFctReturnConfMessage:=2;
	END_CASE
END_FUNCTION

(* POU PRG_VISU_LAYER5/FB_VISU/FB_CTRLEBUTTON, ST *)
FUNCTION_BLOCK FB_CTRLEBUTTON
VAR_INPUT
	xHWStart:BOOL;							(* external start button *)
	xHWStop:BOOL;							(* external stop button *)
	dwActualPage:DWORD;					(* active number page of the visualisation *)
	T_VisuQVis:ST_QVIS;						(* data structure of the visualisation *)
	T_ExchgParam:ST_QVIS_EXCHG_PARAM;	(* data structure of the visualisation *)
	IxSafetyCircuitOn1:BOOL;					(* state of current if it is on or off from the channel 1 *)
	IxSafetyCircuitOn2:BOOL;					(* state of current if it is on or off from the channel 2 *)
END_VAR
VAR_OUTPUT
END_VAR
VAR_IN_OUT
	T_StartButton: ST_BUTTON;				(* data structure of the control button start *)
	T_StopButton:ST_BUTTON;				(* data structure of the control button stop *)
END_VAR
VAR
(* Init. variable *)
	xFirstExecution:BOOL:=FALSE;
(* Variable *)
	iIndexActivPage:INT;
	dwOldActualPage:DWORD;
(* FB Mask *)
	xMaskPageBtStart:BOOL;
	xMaskPageBtStop:BOOL;
(* Trigger *)
	RisingEdgeSignalStartButton:R_TRIG;
	RisingEdgeStartState:R_TRIG;
	RisingEdgeCfgBtStart:R_TRIG;
	RisingEdgeSignalStopButton:R_TRIG;
	RisingEdgeFlagStopProcess:R_TRIG;
(* Tmp variable *)
	xTmp:BOOL;
	(*RisingEdgeConfirmMessage: R_TRIG; *)
END_VAR
(****************************************************************************************************************************************************)
(***********             This Functionblock manage the external start and stop butto, also for the lamp of this button                  ************)
(****************************************************************************************************************************************************)
(* First execution *)
	IF NOT xFirstExecution THEN
		dwOldActualPage:=16#FFFFFFFF;
		RisingEdgeSignalStartButton(CLK:=FALSE);
		RisingEdgeStartState(CLK:=FALSE);
		RisingEdgeCfgBtStart(CLK:=FALSE);
		RisingEdgeSignalStopButton(CLK:=FALSE);
		RisingEdgeFlagStopProcess(CLK:=FALSE);
		(* Set first execution *)
		xFirstExecution:=TRUE;
	END_IF

(* exit FB if Qvis inactiv *)
	IF NOT(T_VisuQVis.T_CtrleVisu.xQvis) THEN RETURN; END_IF
	IF (dwActualPage < 1) OR (dwActualPage > 999) THEN RETURN; END_IF;

(* Index Activ Page *)
	IF dwActualPage = 0 THEN iIndexActivPage:=1;
	ELSE iIndexActivPage:=T_VisuQVis.T_PageIndex[dwActualPage].iIndexConfigPage; END_IF

(* Start Button *)
	xMaskPageBtStart:=FALSE;
	CASE dwActualPage OF
	(* Auto Geometry page *)
	10:	xTmp:=TRUE;
		IF xTmp AND (NOT(IxSafetyCircuitOn1) OR NOT(IxSafetyCircuitOn2)) THEN
			xTmp:=FALSE;	(* Energieversorgung muss eingeschaltet sein *)
		END_IF;
		IF xTmp AND ((T_ExchgParam.T_SafetyCtrl.bStateMessageError <> 0) OR (T_ExchgParam.T_SafetyCtrl.bStateMessageInfo <> 0)) THEN
			xTmp:=FALSE;
		END_IF;
		IF (T_ExchgParam.T_Visu.T_Message.iState = 401) OR (T_ExchgParam.T_Visu.T_Message.iState = 118) OR (T_ExchgParam.T_Visu.T_Message.iState = 119) OR (T_ExchgParam.T_Visu.T_Message.iState = 108) THEN
			xTmp:=FALSE;
		END_IF;
		(* copy state *)
		xMaskPageBtStart:=xTmp;
	(* Auto Groove page *)
	20:	xTmp:=TRUE;
		IF xTmp AND (NOT(IxSafetyCircuitOn1) OR NOT(IxSafetyCircuitOn2)) THEN
			xTmp:=FALSE;	(* Energieversorgung muss eingeschaltet sein *)
		END_IF;
		IF xTmp AND ((T_ExchgParam.T_SafetyCtrl.bStateMessageError <> 0) OR (T_ExchgParam.T_SafetyCtrl.bStateMessageInfo <> 0)) THEN
			xTmp:=FALSE;
		END_IF;
		IF (T_ExchgParam.T_Visu.T_Message.iState = 401) OR (T_ExchgParam.T_Visu.T_Message.iState = 118) OR (T_ExchgParam.T_Visu.T_Message.iState = 119) OR (T_ExchgParam.T_Visu.T_Message.iState = 108) THEN
			xTmp:=FALSE;
		END_IF;
		(* copy state *)
		xMaskPageBtStart:=xTmp;
	(* Reference page *)
	30:	xTmp:=TRUE;
		IF xTmp AND (NOT(IxSafetyCircuitOn1) OR NOT(IxSafetyCircuitOn2)) THEN
			xTmp:=FALSE;	(* Energieversorgung muss eingeschaltet sein *)
		END_IF;
		IF xTmp AND ((T_ExchgParam.T_SafetyCtrl.bStateMessageError <> 0) OR (T_ExchgParam.T_SafetyCtrl.bStateMessageInfo <> 0)) THEN
			xTmp:=FALSE;
		END_IF;
		IF (T_ExchgParam.T_Visu.T_Message.iState = 401) OR (T_ExchgParam.T_Visu.T_Message.iState = 118) OR (T_ExchgParam.T_Visu.T_Message.iState = 119) THEN
			xTmp:=FALSE;
		END_IF;
		IF (T_ExchgParam.T_StationCommon.iConfigMachineType = 1) THEN
			xTmp:=FALSE;
		END_IF;
		(* copy state *)
		xMaskPageBtStart:=xTmp;
	(* Tool Calibration page *)
	110:	xTmp:=TRUE;
		IF xTmp AND (NOT(IxSafetyCircuitOn1) OR NOT(IxSafetyCircuitOn2)) THEN
			xTmp:=FALSE;	(* Energieversorgung muss eingeschaltet sein *)
		END_IF;
		IF xTmp AND ((T_ExchgParam.T_SafetyCtrl.bStateMessageError <> 0) OR (T_ExchgParam.T_SafetyCtrl.bStateMessageInfo <> 0)) THEN
			xTmp:=FALSE;
		END_IF;
		IF (T_ExchgParam.T_Visu.T_Message.iState = 401) OR (T_ExchgParam.T_Visu.T_Message.iState = 118) OR (T_ExchgParam.T_Visu.T_Message.iState = 119) OR
		     (T_ExchgParam.T_Visu.T_Message.iState = 108) THEN
			xTmp:=FALSE;
		END_IF;
		IF ((T_ExchgParam.T_Machine.T_Process.wState AND 16#6) = 16#2) THEN
			xTmp:=FALSE;
		END_IF;
		IF T_ExchgParam.T_FunctionCommon.xOpenOverlayMeasureInput OR T_ExchgParam.T_FunctionCommon.xOpenOverlaySetGrindPlunge THEN
			xTmp:=FALSE;
		END_IF;
		(* copy state *)
		xMaskPageBtStart:=xTmp;
	(* Teach-in Tool Rotation page *)
	210:	xTmp:=	((T_ExchgParam.T_StationCommon.bStateMachine AND 16#7) = 16#1);
		IF xTmp AND (NOT(IxSafetyCircuitOn1) OR NOT(IxSafetyCircuitOn2)) THEN
			xTmp:=FALSE;	(* Energieversorgung muss eingeschaltet sein *)
		END_IF;
		IF xTmp AND ((T_ExchgParam.T_SafetyCtrl.bStateMessageError <> 0) OR (T_ExchgParam.T_SafetyCtrl.bStateMessageInfo <> 0)) THEN
			xTmp:=FALSE;
		END_IF;
		IF (T_ExchgParam.T_Visu.T_Message.iState = 401) OR (T_ExchgParam.T_Visu.T_Message.iState = 118) OR (T_ExchgParam.T_Visu.T_Message.iState = 119) OR
		     (T_ExchgParam.T_Visu.T_Message.iState = 101) THEN
			xTmp:=FALSE;
		END_IF;
		IF (T_ExchgParam.T_TeachIn.iSelectAxisToolRotation = 1) AND xTmp THEN
			IF ((T_ExchgParam.T_StationCommon.bStateAxisReelLeft AND 16#2) = 16#2) THEN
				xTmp:=FALSE;
			END_IF;
		END_IF;
		IF (T_ExchgParam.T_TeachIn.iSelectAxisToolRotation = 2) AND xTmp THEN
			IF ((T_ExchgParam.T_StationCommon.bStateAxisReelCenter AND 16#2) = 16#2) THEN
				xTmp:=FALSE;
			END_IF;
		END_IF;
		IF (T_ExchgParam.T_TeachIn.iSelectAxisToolRotation = 3) AND xTmp THEN
			IF ((T_ExchgParam.T_StationCommon.bStateAxisReelRight AND 16#2) = 16#2) THEN
				xTmp:=FALSE;
			END_IF;
		END_IF;
		(* copy state *)
		xMaskPageBtStart:=xTmp;
	(* Tool Torque page *)
	220:	xTmp:=	((T_ExchgParam.T_StationCommon.bStateMachine AND 16#7) = 16#1);
		IF xTmp AND (NOT(IxSafetyCircuitOn1) OR NOT(IxSafetyCircuitOn2)) THEN
			xTmp:=FALSE;	(* Energieversorgung muss eingeschaltet sein *)
		END_IF;
		IF xTmp AND ((T_ExchgParam.T_SafetyCtrl.bStateMessageError <> 0) OR (T_ExchgParam.T_SafetyCtrl.bStateMessageInfo <> 0)) THEN
			xTmp:=FALSE;
		END_IF;
		IF (T_ExchgParam.T_Visu.T_Message.iState = 401) OR (T_ExchgParam.T_Visu.T_Message.iState = 118) OR (T_ExchgParam.T_Visu.T_Message.iState = 119) OR
		     (T_ExchgParam.T_Visu.T_Message.iState = 101) THEN
			xTmp:=FALSE;
		END_IF;
		IF ((T_ExchgParam.T_StationCommon.bStateAxisReelLeft AND 16#2) = 16#2) THEN
			xTmp:=FALSE;
		END_IF;
		(* copy state *)
		xMaskPageBtStart:=xTmp;
	(* Teach-in Tool Feeder page *)
	310:	xTmp:=	xTmp:=	((T_ExchgParam.T_StationCommon.bStateMachine AND 16#7) = 16#1);
		IF xTmp AND (NOT(IxSafetyCircuitOn1) OR NOT(IxSafetyCircuitOn2)) THEN
			xTmp:=FALSE;	(* Energieversorgung muss eingeschaltet sein *)
		END_IF;
		IF xTmp AND ((T_ExchgParam.T_SafetyCtrl.bStateMessageError <> 0) OR (T_ExchgParam.T_SafetyCtrl.bStateMessageInfo <> 0)) THEN
			xTmp:=FALSE;
		END_IF;
		IF (T_ExchgParam.T_Visu.T_Message.iState = 401) OR (T_ExchgParam.T_Visu.T_Message.iState = 118) OR (T_ExchgParam.T_Visu.T_Message.iState = 119) OR
		     (T_ExchgParam.T_Visu.T_Message.iState = 101) OR (T_ExchgParam.T_Visu.T_Message.iState = 18) THEN
			xTmp:=FALSE;
		END_IF;
		IF (T_ExchgParam.T_TeachIn.iSelectAxisWireFeeder = 1) AND xTmp THEN
			IF ((T_ExchgParam.T_StationCommon.bStateAxisWireFeeder AND 16#2) = 16#2) THEN
				xTmp:=FALSE;
			END_IF;
		END_IF;
		(* copy state *)
		xMaskPageBtStart:=xTmp;
	(* Teach-in Tool Feeder page *)
	330:	xTmp:=	xTmp:=	((T_ExchgParam.T_StationCommon.bStateMachine AND 16#7) = 16#1);
		IF xTmp AND (NOT(IxSafetyCircuitOn1) OR NOT(IxSafetyCircuitOn2)) THEN
			xTmp:=FALSE;	(* Energieversorgung muss eingeschaltet sein *)
		END_IF;
		IF xTmp AND ((T_ExchgParam.T_SafetyCtrl.bStateMessageError <> 0) OR (T_ExchgParam.T_SafetyCtrl.bStateMessageInfo <> 0)) THEN
			xTmp:=FALSE;
		END_IF;
		IF (T_ExchgParam.T_Visu.T_Message.iState = 401) OR (T_ExchgParam.T_Visu.T_Message.iState = 118) OR (T_ExchgParam.T_Visu.T_Message.iState = 119) OR
		     (T_ExchgParam.T_Visu.T_Message.iState = 101) OR (T_ExchgParam.T_Visu.T_Message.iState = 18) THEN
			xTmp:=FALSE;
		END_IF;
		IF (T_ExchgParam.T_TeachIn.iSelectAxisWireFeeder = 1) AND xTmp THEN
			IF ((T_ExchgParam.T_StationCommon.bStateAxisWireFeeder AND 16#2) = 16#2) THEN
				xTmp:=FALSE;
			END_IF;
		END_IF;
		(* copy state *)
		xMaskPageBtStart:=xTmp;
	(* Teach-in Grind Feeder page *)
	410:	xTmp:=	xTmp:=	((T_ExchgParam.T_StationCommon.bStateMachine AND 16#7) = 16#1);
		IF xTmp AND (NOT(IxSafetyCircuitOn1) OR NOT(IxSafetyCircuitOn2)) THEN
			xTmp:=FALSE;	(* Energieversorgung muss eingeschaltet sein *)
		END_IF;
		IF xTmp AND ((T_ExchgParam.T_SafetyCtrl.bStateMessageError <> 0) OR (T_ExchgParam.T_SafetyCtrl.bStateMessageInfo <> 0)) THEN
			xTmp:=FALSE;
		END_IF;
		IF (T_ExchgParam.T_Visu.T_Message.iState = 401) OR (T_ExchgParam.T_Visu.T_Message.iState = 118) OR (T_ExchgParam.T_Visu.T_Message.iState = 119) OR
		     (T_ExchgParam.T_Visu.T_Message.iState = 101) THEN
			xTmp:=FALSE;
		END_IF;
		IF (T_ExchgParam.T_TeachIn.iSelectAxisGrind = 1) AND xTmp THEN
			IF ((T_ExchgParam.T_StationCommon.bStateAxisGrind AND 16#2) = 16#2) THEN
				xTmp:=FALSE;
			END_IF;
		END_IF;
		IF (T_ExchgParam.T_TeachIn.iSelectAxisGrind = 2) AND xTmp THEN
			IF ((T_ExchgParam.T_StationCommon.bStateAxisGrindSpindle AND 16#2) = 16#2) THEN
				xTmp:=FALSE;
			END_IF;
		END_IF;
		(* copy state *)
		xMaskPageBtStart:=xTmp;
	END_CASE

	(* Set state button start *)
	RisingEdgeSignalStartButton(CLK:=xHWStart);
	IF RisingEdgeSignalStartButton.Q THEN T_StartButton.xInputState:=TRUE; ELSE T_StartButton.xInputState:=FALSE; END_IF
	T_StartButton.xInputState:=T_StartButton.xInputState AND T_VisuQVis.T_ConfigPage[iIndexActivPage].xMaskBtStart;

	(* if page change => init. trigger *)
	IF dwActualPage <> dwOldActualPage THEN
		RisingEdgeStartState(CLK:=FALSE);
		RisingEdgeCfgBtStart(CLK:=FALSE);
		(* save value *)
		dwOldActualPage:=dwActualPage;
	END_IF

	(* Led off if action is starting *)
	RisingEdgeStartState(CLK:=T_StartButton.xInputState);
	IF RisingEdgeStartState.Q THEN T_StartButton.xLedState:=FALSE; END_IF
	RisingEdgeCfgBtStart(CLK:=xMaskPageBtStart);
	IF RisingEdgeCfgBtStart.Q THEN T_StartButton.xLedState:=TRUE; END_IF
	T_StartButton.xLedState:=T_StartButton.xLedState AND T_VisuQVis.T_ConfigPage[iIndexActivPage].xMaskBtStart;

	(* set page mask *)
	T_StartButton.xInputState:=T_StartButton.xInputState AND xMaskPageBtStart;
	T_StartButton.xLedState:=T_StartButton.xLedState AND xMaskPageBtStart;

(* Stop Button *)
	xMaskPageBtStop:=FALSE;
	RisingEdgeSignalStopButton(CLK:=xHWStop);
	IF RisingEdgeSignalStopButton.Q THEN T_StopButton.xInputState:=TRUE; ELSE T_StopButton.xInputState:=FALSE; END_IF
	T_StopButton.xInputState:=T_StopButton.xInputState AND T_VisuQVis.T_ConfigPage[iIndexActivPage].xMaskBtStop;
	T_StopButton.xLedState:=T_VisuQVis.T_ConfigPage[iIndexActivPage].xMaskBtStop;

	(* if machine process inactiv => set mask inactiv *)
	IF dwActualPage > 0 THEN
		IF (T_ExchgParam.T_Machine.T_Process.wState AND 16#14) = 16#0 THEN
		(* process activ and no error *)
			IF (T_ExchgParam.T_Machine.T_Process.wState AND 16#80) = 16#0 THEN xMaskPageBtStop:=TRUE; ELSE xMaskPageBtStop:=FALSE; END_IF
		ELSIF ((dwActualPage = 210) OR (dwActualPage = 310) OR (dwActualPage = 410)) THEN
			(* Achse muss Aktiv sein, Stationsendflag muss gesetzt sein, Prozessendflag muss gesetzt sein *)
			IF ((T_ExchgParam.T_StationCommon.bStateMachine AND 16#7) = 16#3) AND ((T_ExchgParam.T_Machine.T_Process.wState AND 16#2) = 16#0) THEN
				xMaskPageBtStop:=TRUE;
			END_IF;
			(* Achse darf nicht Aktiv sein, Stationsendflag muss gesetzt sein,  Prozessendflag muss gesetzt sein *)
			IF ((T_ExchgParam.T_StationCommon.bStateMachine AND 16#7) = 16#1) AND ((T_ExchgParam.T_Machine.T_Process.wState AND 16#2) = 16#0) THEN
				xMaskPageBtStop:=FALSE;
				IF (T_ExchgParam.T_TeachIn.iSelectAxisToolRotation = 1) AND (dwActualPage = 210) THEN
					IF ((T_ExchgParam.T_StationCommon.bStateAxisReelLeft AND 16#2) = 16#2) THEN
						xMaskPageBtStop:=TRUE;
					END_IF;
				END_IF;
				IF (T_ExchgParam.T_TeachIn.iSelectAxisToolRotation = 2) AND (dwActualPage = 210) THEN
					IF ((T_ExchgParam.T_StationCommon.bStateAxisReelCenter AND 16#2) = 16#2) THEN
						xMaskPageBtStop:=TRUE;
					END_IF;
				END_IF;
				IF (T_ExchgParam.T_TeachIn.iSelectAxisToolRotation = 3) AND (dwActualPage = 210) THEN
					IF ((T_ExchgParam.T_StationCommon.bStateAxisReelRight AND 16#2) = 16#2) THEN
						xMaskPageBtStop:=TRUE;
					END_IF;
				END_IF;
				IF (T_ExchgParam.T_TeachIn.iSelectAxisWireFeeder = 1) AND (dwActualPage = 310) THEN
					IF ((T_ExchgParam.T_StationCommon.bStateAxisWireFeeder AND 16#2) = 16#2) THEN
						xMaskPageBtStop:=TRUE;
					END_IF;
				END_IF;
				IF (T_ExchgParam.T_TeachIn.iSelectAxisGrind = 1) AND (dwActualPage = 410) THEN
					IF ((T_ExchgParam.T_StationCommon.bStateAxisGrind AND 16#2) = 16#2) THEN
						xMaskPageBtStop:=TRUE;
					END_IF;
				END_IF;
				IF (T_ExchgParam.T_TeachIn.iSelectAxisGrind = 2) AND (dwActualPage = 410) THEN
					IF ((T_ExchgParam.T_StationCommon.bStateAxisGrindSpindle AND 16#2) = 16#2) THEN
						xMaskPageBtStop:=TRUE;
					END_IF;
				END_IF;
			END_IF;
			IF (T_VisuQVis.T_CtrleAction.iFunction = 301) AND NOT(T_VisuQVis.T_CtrleAction.xDone) THEN
				xMaskPageBtStop:=FALSE;
			END_IF;
		ELSIF (dwActualPage = 220) THEN
			(* Achse muss Aktiv sein, Stationsendflag muss gesetzt sein, Prozessendflag muss gesetzt sein *)
			xMaskPageBtStop:=FALSE;
			IF ((T_ExchgParam.T_StationCommon.bStateAxisReelLeft AND 16#2) = 16#2) THEN
				xMaskPageBtStop:=TRUE;
			END_IF;
			IF (T_VisuQVis.T_CtrleAction.iFunction = 403) AND NOT(T_VisuQVis.T_CtrleAction.xDone) THEN
				xMaskPageBtStop:=FALSE;
			END_IF;
		(* process inactiv *)
		ELSE xMaskPageBtStop:=FALSE; END_IF
		IF (T_ExchgParam.T_Visu.T_Message.iState = 401) OR (T_ExchgParam.T_Visu.T_Message.iState = 118) OR (T_ExchgParam.T_Visu.T_Message.iState = 119) THEN
			xMaskPageBtStop:=FALSE;
		END_IF;
		IF NOT(IxSafetyCircuitOn1) OR NOT(IxSafetyCircuitOn2) THEN
			xMaskPageBtStop:=FALSE;
		END_IF;
	END_IF

	(* set page mask *)
	T_StopButton.xInputState:=T_StopButton.xInputState AND xMaskPageBtStop;
	T_StopButton.xLedState:=T_StopButton.xLedState AND xMaskPageBtStop;
END_FUNCTION_BLOCK

(* POU PRG_VISU_LAYER5/FB_VISU/xFctCtrleProfileName, ST *)
FUNCTION xFctCtrleProfileName : BOOL
VAR_INPUT
	sNewProfileName:STRING(30);		(* profile name to save *)
	ptrProfileList:POINTER TO ARRAY[1..csiMaxProfile] OF ST_PROFILE_ID;	(* list of the saved profil names *)
END_VAR
VAR
(* variable *)
	i: INT;
	sTmp:STRING;
	sTmp2:STRING;
END_VAR
(****************************************************************************************************************************************************)
(***********                                              This Function check the name of the profile if it is correct                                                     ************)
(****************************************************************************************************************************************************)
(* Init. function *)
	xFctCtrleProfileName:=FALSE;
	sTmp:=FCT_UPLOW_CASE(	xLowConvert:=TRUE,
							sInString:=sNewProfileName);

(* Search if name already exists *)
	FOR i:=1 TO csiMaxProfile DO
		sTmp2:=	FCT_UPLOW_CASE(	xLowConvert:=TRUE,
								sInString:=ptrProfileList^[i].sName);
		IF sTmp = sTmp2 AND sTmp2 <> '' THEN RETURN; END_IF
	END_FOR

(* Confirm function *)
	xFctCtrleProfileName:=TRUE;
END_FUNCTION

(* POU GENERAL/FCT_UPLOW_CASE, ST *)
FUNCTION FCT_UPLOW_CASE : STRING
VAR_INPUT
	xLowConvert:BOOL;			(* FALSE=conversion to up case, TRUE=conversion in low case *)
	sInString:STRING;				(* string with 80 character, which will be convert *)
END_VAR
VAR
(* variable *)
	sListUpCase:STRING:='ABCDEFGHIJKLMNOPQRSTUVWXYZ';
	sListLowCase:STRING:='abcdefghijklmnopqrstuvwxyz';
	i:INT;
(* Tmp *)
	sTmp:STRING;
	iTmp:INT;
END_VAR
(****************************************************************************************************************************************************)
(***********                                                      This function convert a String in up or low case                                                                ************)
(****************************************************************************************************************************************************)
(* Init. *)
	FCT_UPLOW_CASE:='';

(*Test string size*)
	IF LEN(sInString) < 1 OR LEN(sInString) > 255 THEN RETURN; END_IF

	IF xLowConvert THEN
	(* Conversion to low case *)
		FOR i:= 1 TO LEN(sInString) DO
			sTmp:=MID(sInString,1,i);
			iTmp:=FIND(sListUpCase,sTmp);
			IF iTmp > 0 THEN FCT_UPLOW_CASE:=CONCAT(FCT_UPLOW_CASE,MID(sListLowCase,1,iTmp));
				ELSE FCT_UPLOW_CASE:=CONCAT(FCT_UPLOW_CASE,sTmp); END_IF
		END_FOR
	(* Conversion to up case *)
	ELSE
		FOR i:= 1 TO LEN(sInString) DO
			sTmp:=MID(sInString,1,i);
			iTmp:=FIND(sListLowCase,sTmp);
			IF iTmp > 0 THEN FCT_UPLOW_CASE:=CONCAT(FCT_UPLOW_CASE,MID(sListUpCase,1,iTmp));
				ELSE FCT_UPLOW_CASE:=CONCAT(FCT_UPLOW_CASE,sTmp); END_IF
		END_FOR
	END_IF
END_FUNCTION

(* POU PRG_VISU_LAYER5/FB_VISU/iFctExistProfileName, ST *)
FUNCTION iFctExistProfileName : INT
VAR_INPUT
	sProfileName:STRING(30);											(* name of the profile, which will be saved *)
	ptrProfileList:POINTER TO ARRAY[1..csiMaxProfile] OF ST_PROFILE_ID;	(* list of profil names which are saved *)
END_VAR
VAR
	i:INT;
	sTmp:STRING;
	sTmp2:STRING;
END_VAR
(****************************************************************************************************************************************************)
(***********                                               This Function check if the name of the profile already exists                                              ************)
(****************************************************************************************************************************************************)
(* Init. function *)
	iFctExistProfileName:=0;
	sTmp:=FCT_UPLOW_CASE(	xLowConvert:=TRUE,
							sInString:=sProfileName);

(* Search if name already exists *)
	FOR i:=1 TO csiMaxProfile DO
		sTmp2:=	FCT_UPLOW_CASE(	xLowConvert:=TRUE,
								sInString:=ptrProfileList^[i].sName);
		IF sTmp = sTmp2 AND sTmp2 <> '' THEN iFctExistProfileName:=i; RETURN; END_IF
	END_FOR
END_FUNCTION

(* POU PRG_PROCESS_LAYER4/PRG_PROCESS, FBD *)
PROGRAM PRG_PROCESS
VAR
	FBProcess: FB_PROCESS;
	xReady: BOOL;
	xEnd: BOOL;
	xStop: BOOL;
	xReferenced: BOOL;
	xError: BOOL;
	iErrorNr: DINT;
	iFunctionNr: INT;
END_VAR
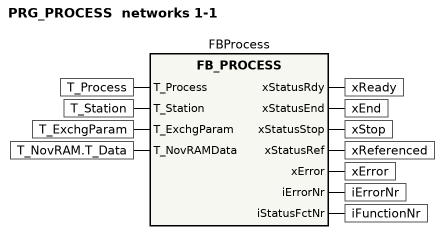
_FBD_ (* Function Block Diagram *)
NETWORK 1 (* PROCESS LEVEL-->LAYER 4 *)
	FBProcess:FB_PROCESS(T_Process: T_Process, T_Station: T_Station, T_ExchgParam: T_ExchgParam, T_NovRAMData: T_NovRAM.T_Data, xStatusEnd => xEnd, xStatusStop => xStop, xStatusRef => xReferenced, xError => xError, iErrorNr => iErrorNr, iStatusFctNr => iFunctionNr) => xReady
_END_FBD_
(* the same logic as Structured Text *)
(* Network 1: PROCESS LEVEL-->LAYER 4 *)
FBProcess(T_Process := T_Process, T_Station := T_Station, T_ExchgParam := T_ExchgParam, T_NovRAMData := T_NovRAM.T_Data);
xEnd := FBProcess.xStatusEnd;
xStop := FBProcess.xStatusStop;
xReferenced := FBProcess.xStatusRef;
xError := FBProcess.xError;
iErrorNr := FBProcess.iErrorNr;
iFunctionNr := FBProcess.iStatusFctNr;
xReady := FBProcess.xStatusRdy;
END_PROGRAM

(* POU PRG_PROCESS_LAYER4/FB_PROCESS/FB_PROCESS, ST *)
FUNCTION_BLOCK FB_PROCESS
VAR_INPUT
END_VAR
VAR_IN_OUT
	T_Process : ST_PROCESS;				(* data structure of the processlevel *)
	T_Station : ST_STATION;					(* data structure of the stationlevel *)
	T_ExchgParam:ST_QVIS_EXCHG_PARAM;	(* data structure of the visualisation *)
	T_NovRAMData:ST_DATA_RETAIN;		(* data structure of the NovRam *)
END_VAR
VAR_OUTPUT
	xStatusRdy : BOOL := FALSE;				(* state of the processlevel if it is ready or not *)
	xStatusEnd : BOOL := FALSE;				(* state of the processlevel if a process is active or not *)
	xStatusStop : BOOL := FALSE;				(* state of the processlevel if a process will be stopped *)
	xStatusRef : BOOL := FALSE;				(* state of the processlevel if the machine is referenced *)
	xError : BOOL := FALSE;					(* state of the processlevel if the machine has an error *)
	iErrorNr : DINT :=0;							(* state of the processlevel if the machine has an error, in this case it will give the errornumber *)
	iStatusFctNr : INT := 0;						(* state of the processlevel, which process is active *)
END_VAR
VAR
	xStartFunction: BOOL;
	xSetEnd: BOOL;
	iPrcFunctionNr: INT;
	xProcessError: BOOL;
	xInitError: BOOL;
	xTmpStart: BOOL;
	xInitStart: BOOL;
	xInitStop: BOOL;
	xTmpStopFunction: BOOL;
	xDisable: BOOL;
	xResetRef: BOOL;
	xInitStopCycle: BOOL;
	xTmpStopCycleFunction: BOOL;
(* end modif test torque *)
	FBErrorMessage : FB_ErrorMessage;
	FBPrcMachineReference: FB_PrcMachineReference;
	FBPrcAutoGeometry: FB_PrcAutoGeometry;
	diTmpErrorNr: DINT;
	xResetAutoGeometry: BOOL;
	FBPrcAutoGroove: FB_PrcAutoGroove;
	xResetAutoGroove: BOOL;
	FBPrcToolCalibration: FB_PrcToolCalibration;
	xResetToolCalibration: BOOL;
END_VAR
(****************************************************************************************************************************************************)
(***********                                            This Functionblock manage all the machine process                                                             ************)
(****************************************************************************************************************************************************)
IF NOT(T_Process.xEnable) THEN
	T_Process.xRdy:=FALSE;
	xDisable:=TRUE;
	RETURN;
ELSE
	IF xDisable THEN
		T_Process.xRdy:=TRUE;
		xDisable:=FALSE;
		xSetEnd:=TRUE;
	END_IF;
END_IF;
(******************************************************************************************************************************************)
(****************************				                  Status Part                                                            *****************************)
(******************************************************************************************************************************************)
xStatusRdy:=T_Process.xRdy;
xStatusEnd:=T_Process.xEnd;
xStatusRef:=T_Station.TControl.xReferenced;
T_Process.xReferenced:=xStatusRef;
xError:=T_Process.xError;
iStatusFctNr:=iPrcFunctionNr;


